	    // Counter hanya jalan saat tidak sedang sequence reset/release
	    IF #SeqMco = 0 THEN
	        IF "Win".Msc.Mco.Act < "Win".Msc.Mco.Set THEN
	            "Win".Msc.Mco.Act := "Win".Msc.Mco.Act + #McoStep;

	            IF "Win".Msc.Mco.Act >= "Win".Msc.Mco.Set THEN
	                "Win".Msc.Mco.Act := "Win".Msc.Mco.Set;
	                #McoReachedLatch := TRUE;
	            END_IF;
	        END_IF;
	    END_IF;

	    // Remaining meter
	    #McoRemain := "Win".Msc.Mco.Set - "Win".Msc.Mco.Act;
	    IF #McoRemain < 0.0 THEN
	        #McoRemain := 0.0;
	    END_IF;

	    // Time remaining dalam menit
	    IF #LineSpd > 0.0 THEN
	        "Win".Msc.Mco.Tim := #McoRemain / #LineSpd;
	    ELSE
	        "Win".Msc.Mco.Tim := 0.0;
	    END_IF;

	    // Trigger sequence jika setpoint tercapai
	    IF (#McoReachedLatch) AND (#SeqMco = 0) THEN
	        #McoReachedLatch := FALSE;
	        #SeqMco := 1;
	    END_IF;

	    // Sequential pulse:
	    // step 1 : Rst TRUE
	    // step 2 : Rst FALSE, Rel TRUE, reset Act ke 0
	    // step 0 : semua FALSE
	    CASE #SeqMco OF
	        0:
	            ;
	        1:
	            "Win".Msc.Mco.Rst := TRUE;
	            #SeqMco := 2;

	        2:
	            "Win".Msc.Mco.Rel := TRUE;
	            "Win".Msc.Mco.Act := 0.0;
	            #SeqMco := 0;
	        ELSE
	            #SeqMco := 0;
	    END_CASE;

	    "Win".Msc.AutCycTim.Act := "FC_NoiseReal"(Base := 300.0, Amp := #Amp_PosMm, Lo := #Lo, Hi := #Hi, Seed := #Seed);

	    // =========================
	    // WINDER 1 & 2
	    // =========================
	    "Win".W01.Drv.SpdSet := "FC_NoiseReal"(Base := 177.7, Amp := #Amp_SpdMpm, Lo := #Lo, Hi := #Hi, Seed := #Seed);
	    "Win".W01.Drv.SpdAct := "FC_NoiseReal"(Base := 171.2, Amp := #Amp_SpdMpm, Lo := #Lo, Hi := #Hi, Seed := #Seed);
	    "Win".W01.Drv.LoaAct := "FC_NoiseReal"(Base := 10.3, Amp := #Amp_LoaPct, Lo := #Lo, Hi := #Hi, Seed := #Seed);
	    "Win".W01.Gbl.TenSet := "FC_NoiseReal"(Base := 232.4, Amp := #Amp_TenNm, Lo := #Lo, Hi := #Hi, Seed := #Seed);
	    "Win".W01.Gbl.ScwTenSet := "FC_NoiseReal"(Base := 15.0, Amp := #Amp_LoaPct, Lo := #Lo, Hi := #Hi, Seed := #Seed);
	    "Win".W01.Prs.SetAct := "FC_NoiseReal"(Base := 1059.0, Amp := #Amp_PrsN, Lo := #Lo, Hi := #Hi, Seed := #Seed);
	    "Win".W01.Dia.Act := "FC_NoiseReal"(Base := 576.0, Amp := #Amp_PosMm, Lo := #Lo, Hi := #Hi, Seed := #Seed);

	    "Win".W02.Drv.SpdSet := "FC_NoiseReal"(Base := 0.0, Amp := #Amp_SpdMpm, Lo := #Lo, Hi := #Hi, Seed := #Seed);
	    "Win".W02.Drv.SpdAct := "FC_NoiseReal"(Base := 0.0, Amp := #Amp_SpdMpm, Lo := #Lo, Hi := #Hi, Seed := #Seed);
	    "Win".W02.Drv.LoaAct := "FC_NoiseReal"(Base := 0.0, Amp := #Amp_LoaPct, Lo := #Lo, Hi := #Hi, Seed := #Seed);
	    "Win".W02.Gbl.TenSet := "FC_NoiseReal"(Base := 234.4, Amp := #Amp_TenNm, Lo := #Lo, Hi := #Hi, Seed := #Seed);
	    "Win".W02.Gbl.ScwTenSet := "FC_NoiseReal"(Base := 15.0, Amp := #Amp_LoaPct, Lo := #Lo, Hi := #Hi, Seed := #Seed);
	    "Win".W02.Prs.SetAct := "FC_NoiseReal"(Base := 1056.0, Amp := #Amp_PrsN, Lo := #Lo, Hi := #Hi, Seed := #Seed);
	    "Win".W02.Dia.Act := "FC_NoiseReal"(Base := 0.0, Amp := #Amp_PosMm, Lo := #Lo, Hi := #Hi, Seed := #Seed);

END_FUNCTION_BLOCK

FUNCTION "FC_Fluct_DB325_StrTdoOut" : Void
{ S7_Optimized_Access := 'TRUE' }
VERSION : 0.1
// ============================================================
// FLUCTUATION DB325 (StrTdoOut) - TDO Outlet
// ============================================================
   VAR_INPUT
      Enable : Bool;   // amplitudo fluktuasi
      Amp_TmpC : Real;   // Â±Â°C
      Amp_Y_Pct : Real;   // Â±%
      Amp_SpdMpm : Real;   // Â± m/min
      Amp_Loa_Pct : Real;   // Â± %
   END_VAR

   VAR_IN_OUT
      Seed : DInt;
   END_VAR

   VAR_TEMP
      Lo : Real;
      Hi : Real;
   END_VAR


BEGIN
	    IF NOT #Enable THEN
	        RETURN;
	    END_IF;

	    #Lo := -3.4E38;
	    #Hi := 3.4E38;

	    // -------------------------
	    // Drive TDO Outlet (Drv001)
	    // -------------------------
	    "StrTdoOut".Drv001.SpdSet := "FC_NoiseReal"(Base := 175.0, Amp := #Amp_SpdMpm, Lo := #Lo, Hi := #Hi, Seed := #Seed);
	    "StrTdoOut".Drv001.SpdAct := "FC_NoiseReal"(Base := 175.0, Amp := #Amp_SpdMpm, Lo := #Lo, Hi := #Hi, Seed := #Seed);
	    "StrTdoOut".Drv001.LoaAct := "FC_NoiseReal"(Base := 20.8, Amp := #Amp_Loa_Pct, Lo := #Lo, Hi := #Hi, Seed := #Seed);

	    // -------------------------
	    // All Zone
	    // -------------------------
	    "StrTdoOut".TmpAll.Set := "FC_NoiseReal"(Base := 145.0, Amp := #Amp_TmpC, Lo := #Lo, Hi := #Hi, Seed := #Seed);

	    // -------------------------
	    // Annealing 1.1 (Ann011)
	    // -------------------------
	    "StrTdoOut".TmpAnn011.Set := "FC_NoiseReal"(Base := 145.0, Amp := #Amp_TmpC, Lo := #Lo, Hi := #Hi, Seed := #Seed);
	    "StrTdoOut".TmpAnn011.Act := "FC_NoiseReal"(Base := 145.1, Amp := #Amp_TmpC, Lo := #Lo, Hi := #Hi, Seed := #Seed);
	    "StrTdoOut".TmpAnn011.Y := "FC_NoiseReal"(Base := 0.0, Amp := #Amp_Y_Pct, Lo := #Lo, Hi := #Hi, Seed := #Seed);

	    // Annealing 1.2 (Ann012)
	    "StrTdoOut".TmpAnn012.Set := "FC_NoiseReal"(Base := 145.0, Amp := #Amp_TmpC, Lo := #Lo, Hi := #Hi, Seed := #Seed);
	    "StrTdoOut".TmpAnn012.Act := "FC_NoiseReal"(Base := 148.1, Amp := #Amp_TmpC, Lo := #Lo, Hi := #Hi, Seed := #Seed);
	    "StrTdoOut".TmpAnn012.Y := "FC_NoiseReal"(Base := 0.0, Amp := #Amp_Y_Pct, Lo := #Lo, Hi := #Hi, Seed := #Seed);

	    // -------------------------
	    // Annealing 2.1 (Ann021)
	    // -------------------------
	    "StrTdoOut".TmpAnn021.Set := "FC_NoiseReal"(Base := 135.0, Amp := #Amp_TmpC, Lo := #Lo, Hi := #Hi, Seed := #Seed);
	    "StrTdoOut".TmpAnn021.Act := "FC_NoiseReal"(Base := 134.7, Amp := #Amp_TmpC, Lo := #Lo, Hi := #Hi, Seed := #Seed);
	    "StrTdoOut".TmpAnn021.Y := "FC_NoiseReal"(Base := 3.0, Amp := #Amp_Y_Pct, Lo := #Lo, Hi := #Hi, Seed := #Seed);

	    // Annealing 2.2 (Ann022)
	    "StrTdoOut".TmpAnn022.Set := "FC_NoiseReal"(Base := 135.0, Amp := #Amp_TmpC, Lo := #Lo, Hi := #Hi, Seed := #Seed);
	    "StrTdoOut".TmpAnn022.Act := "FC_NoiseReal"(Base := 136.2, Amp := #Amp_TmpC, Lo := #Lo, Hi := #Hi, Seed := #Seed);
	    "StrTdoOut".TmpAnn022.Y := "FC_NoiseReal"(Base := 0.0, Amp := #Amp_Y_Pct, Lo := #Lo, Hi := #Hi, Seed := #Seed);

	    // -------------------------
	    // Annealing 3.1 (Ann031)
	    // -------------------------
	    "StrTdoOut".TmpAnn031.Set := "FC_NoiseReal"(Base := 135.0, Amp := #Amp_TmpC, Lo := #Lo, Hi := #Hi, Seed := #Seed);
	    "StrTdoOut".TmpAnn031.Act := "FC_NoiseReal"(Base := 135.1, Amp := #Amp_TmpC, Lo := #Lo, Hi := #Hi, Seed := #Seed);
	    "StrTdoOut".TmpAnn031.Y := "FC_NoiseReal"(Base := 8.0, Amp := #Amp_Y_Pct, Lo := #Lo, Hi := #Hi, Seed := #Seed);

	    // Annealing 3.2 (Ann032)
	    "StrTdoOut".TmpAnn032.Set := "FC_NoiseReal"(Base := 135.0, Amp := #Amp_TmpC, Lo := #Lo, Hi := #Hi, Seed := #Seed);
	    "StrTdoOut".TmpAnn032.Act := "FC_NoiseReal"(Base := 133.5, Amp := #Amp_TmpC, Lo := #Lo, Hi := #Hi, Seed := #Seed);
	    "StrTdoOut".TmpAnn032.Y := "FC_NoiseReal"(Base := 11.0, Amp := #Amp_Y_Pct, Lo := #Lo, Hi := #Hi, Seed := #Seed);

END_FUNCTION

FUNCTION "FC_Fluct_DB323_324_TdoInlMid" : Void
{ S7_Optimized_Access := 'TRUE' }
VERSION : 0.1
// ============================================================
// FLUCTUATION DB323 + DB324
// AREA: StrTdoInl + StrTdoMid
// ============================================================
   VAR_INPUT
      Enable : Bool;   // amplitudo fluktuasi
      Amp_TmpC : Real;   // Â±Â°C
      Amp_Y_Pct : Real;   // Â±%
   END_VAR

   VAR_IN_OUT
      Seed : DInt;
   END_VAR

   VAR_TEMP
      Lo : Real;
      Hi : Real;
   END_VAR


BEGIN
	    IF NOT #Enable THEN
	        RETURN;
	    END_IF;

	    #Lo := -3.4E38;
	    #Hi := 3.4E38;

	    // =====================================================
	    // DB323 - StrTdoInl
	    // =====================================================

	    // All Zone
	    "StrTdoInl".TmpAll.Set := "FC_NoiseReal"(Base := 179.0, Amp := #Amp_TmpC, Lo := #Lo, Hi := #Hi, Seed := #Seed);

	    // Preheating 1
	    "StrTdoInl".TmpPrh001.Set := "FC_NoiseReal"(Base := 164.0, Amp := #Amp_TmpC, Lo := #Lo, Hi := #Hi, Seed := #Seed);
	    "StrTdoInl".TmpPrh001.Act := "FC_NoiseReal"(Base := 164.0, Amp := #Amp_TmpC, Lo := #Lo, Hi := #Hi, Seed := #Seed);
	    "StrTdoInl".TmpPrh001.Y := "FC_NoiseReal"(Base := 35.0, Amp := #Amp_Y_Pct, Lo := #Lo, Hi := #Hi, Seed := #Seed);

	    // Preheating 2
	    "StrTdoInl".TmpPrh002.Set := "FC_NoiseReal"(Base := 174.0, Amp := #Amp_TmpC, Lo := #Lo, Hi := #Hi, Seed := #Seed);
	    "StrTdoInl".TmpPrh002.Act := "FC_NoiseReal"(Base := 173.3, Amp := #Amp_TmpC, Lo := #Lo, Hi := #Hi, Seed := #Seed);
	    "StrTdoInl".TmpPrh002.Y := "FC_NoiseReal"(Base := 100.0, Amp := #Amp_Y_Pct, Lo := #Lo, Hi := #Hi, Seed := #Seed);

	    // Preheating 3
	    "StrTdoInl".TmpPrh003.Set := "FC_NoiseReal"(Base := 179.0, Amp := #Amp_TmpC, Lo := #Lo, Hi := #Hi, Seed := #Seed);
	    "StrTdoInl".TmpPrh003.Act := "FC_NoiseReal"(Base := 179.2, Amp := #Amp_TmpC, Lo := #Lo, Hi := #Hi, Seed := #Seed);
	    "StrTdoInl".TmpPrh003.Y := "FC_NoiseReal"(Base := 20.0, Amp := #Amp_Y_Pct, Lo := #Lo, Hi := #Hi, Seed := #Seed);

	    // =====================================================
	    // DB324 - StrTdoMid
	    // =====================================================

	    // All Zone
	    "StrTdoMid".TmpAll.Set := "FC_NoiseReal"(Base := 157.0, Amp := #Amp_TmpC, Lo := #Lo, Hi := #Hi, Seed := #Seed);

	    // Drawing 1.1
	    "StrTdoMid".TmpDrw011.Set := "FC_NoiseReal"(Base := 157.0, Amp := #Amp_TmpC, Lo := #Lo, Hi := #Hi, Seed := #Seed);
	    "StrTdoMid".TmpDrw011.Act := "FC_NoiseReal"(Base := 157.0, Amp := #Amp_TmpC, Lo := #Lo, Hi := #Hi, Seed := #Seed);
	    "StrTdoMid".TmpDrw011.Y := "FC_NoiseReal"(Base := 54.0, Amp := #Amp_Y_Pct, Lo := #Lo, Hi := #Hi, Seed := #Seed);

	    // Drawing 1.2
	    "StrTdoMid".TmpDrw012.Set := "FC_NoiseReal"(Base := 157.0, Amp := #Amp_TmpC, Lo := #Lo, Hi := #Hi, Seed := #Seed);
	    "StrTdoMid".TmpDrw012.Act := "FC_NoiseReal"(Base := 156.8, Amp := #Amp_TmpC, Lo := #Lo, Hi := #Hi, Seed := #Seed);
	    "StrTdoMid".TmpDrw012.Y := "FC_NoiseReal"(Base := 14.0, Amp := #Amp_Y_Pct, Lo := #Lo, Hi := #Hi, Seed := #Seed);

	    // Drawing 2.1
	    "StrTdoMid".TmpDrw021.Set := "FC_NoiseReal"(Base := 157.0, Amp := #Amp_TmpC, Lo := #Lo, Hi := #Hi, Seed := #Seed);
	    "StrTdoMid".TmpDrw021.Act := "FC_NoiseReal"(Base := 156.9, Amp := #Amp_TmpC, Lo := #Lo, Hi := #Hi, Seed := #Seed);
	    "StrTdoMid".TmpDrw021.Y := "FC_NoiseReal"(Base := 4.0, Amp := #Amp_Y_Pct, Lo := #Lo, Hi := #Hi, Seed := #Seed);

	    // Drawing 2.2
	    "StrTdoMid".TmpDrw022.Set := "FC_NoiseReal"(Base := 157.0, Amp := #Amp_TmpC, Lo := #Lo, Hi := #Hi, Seed := #Seed);
	    "StrTdoMid".TmpDrw022.Act := "FC_NoiseReal"(Base := 157.0, Amp := #Amp_TmpC, Lo := #Lo, Hi := #Hi, Seed := #Seed);
	    "StrTdoMid".TmpDrw022.Y := "FC_NoiseReal"(Base := 2.0, Amp := #Amp_Y_Pct, Lo := #Lo, Hi := #Hi, Seed := #Seed);

	    // Drawing 3.1
	    "StrTdoMid".TmpDrw031.Set := "FC_NoiseReal"(Base := 156.0, Amp := #Amp_TmpC, Lo := #Lo, Hi := #Hi, Seed := #Seed);
	    "StrTdoMid".TmpDrw031.Act := "FC_NoiseReal"(Base := 156.0, Amp := #Amp_TmpC, Lo := #Lo, Hi := #Hi, Seed := #Seed);
	    "StrTdoMid".TmpDrw031.Y := "FC_NoiseReal"(Base := 63.0, Amp := #Amp_Y_Pct, Lo := #Lo, Hi := #Hi, Seed := #Seed);

	    // Drawing 3.2
	    "StrTdoMid".TmpDrw032.Set := "FC_NoiseReal"(Base := 156.0, Amp := #Amp_TmpC, Lo := #Lo, Hi := #Hi, Seed := #Seed);
	    "StrTdoMid".TmpDrw032.Act := "FC_NoiseReal"(Base := 155.8, Amp := #Amp_TmpC, Lo := #Lo, Hi := #Hi, Seed := #Seed);
	    "StrTdoMid".TmpDrw032.Y := "FC_NoiseReal"(Base := 10.0, Amp := #Amp_Y_Pct, Lo := #Lo, Hi := #Hi, Seed := #Seed);

	    // Drawing 4.1
	    "StrTdoMid".TmpDrw041.Set := "FC_NoiseReal"(Base := 155.0, Amp := #Amp_TmpC, Lo := #Lo, Hi := #Hi, Seed := #Seed);
	    "StrTdoMid".TmpDrw041.Act := "FC_NoiseReal"(Base := 154.3, Amp := #Amp_TmpC, Lo := #Lo, Hi := #Hi, Seed := #Seed);
	    "StrTdoMid".TmpDrw041.Y := "FC_NoiseReal"(Base := 3.0, Amp := #Amp_Y_Pct, Lo := #Lo, Hi := #Hi, Seed := #Seed);

	    // Drawing 4.2
	    "StrTdoMid".TmpDrw042.Set := "FC_NoiseReal"(Base := 155.0, Amp := #Amp_TmpC, Lo := #Lo, Hi := #Hi, Seed := #Seed);
	    "StrTdoMid".TmpDrw042.Act := "FC_NoiseReal"(Base := 156.0, Amp := #Amp_TmpC, Lo := #Lo, Hi := #Hi, Seed := #Seed);
	    "StrTdoMid".TmpDrw042.Y := "FC_NoiseReal"(Base := 0.0, Amp := #Amp_Y_Pct, Lo := #Lo, Hi := #Hi, Seed := #Seed);

END_FUNCTION

FUNCTION "FC_Fluct_DB313_ExtFil" : Void
{ S7_Optimized_Access := 'TRUE' }
VERSION : 0.1
// ============================================================
// FLUCTUATION DB313 (ExtFil)
// ============================================================
   VAR_INPUT
      Enable : Bool;   // amplitudo fluktuasi
      Amp_TmpC : Real;   // Â±Â°C
      Amp_PrsBar : Real;   // Â±bar
      Amp_Y_Pct : Real;   // Â±%
   END_VAR

   VAR_IN_OUT
      Seed : DInt;
   END_VAR

   VAR_TEMP
      Lo : Real;
      Hi : Real;
   END_VAR


BEGIN
	    IF NOT #Enable THEN
	        RETURN;
	    END_IF;

	    #Lo := -3.4E38;
	    #Hi := 3.4E38;

	    // =========================
	    // Pressure (S7_PRS) - base dari gambar + comment ExtFil.db
	    // Prs001: before filter  (Press P3 = 97.9 bar)
	    // Prs002: after filter   (Press P2 = 135.6 bar)
	    // Prs012: diff pressure  (Diff Press = 37.7 bar)
	    // Prs003: before die     (Press P4 = 0.0 bar)
	    // =========================
	    "ExtFil".Prs001.Act := "FC_NoiseReal"(Base := 97.9, Amp := #Amp_PrsBar, Lo := #Lo, Hi := #Hi, Seed := #Seed);
	    "ExtFil".Prs002.Act := "FC_NoiseReal"(Base := 135.6, Amp := #Amp_PrsBar, Lo := #Lo, Hi := #Hi, Seed := #Seed);
	    "ExtFil".Prs012.Act := "FC_NoiseReal"(Base := 37.7, Amp := #Amp_PrsBar, Lo := #Lo, Hi := #Hi, Seed := #Seed);
	    "ExtFil".Prs003.Act := "FC_NoiseReal"(Base := 0.0, Amp := #Amp_PrsBar, Lo := #Lo, Hi := #Hi, Seed := #Seed);

	    // =========================
	    // Melt Temp (S7_ACT) - base dari gambar
	    // TmpMel001: before filter (Melt Temp T3 = 241.1 Â°C)
	    // TmpMel002: after filter  (Melt Temp T2 = 244.6 Â°C)
	    // TmpMel003: before die    (Melt Temp T4 = 1999.9 Â°C)  // sesuai tampilan
	    // TmpMel004: preheating filter (Pre.Filter = 32.4 Â°C)
	    // =========================
	    "ExtFil".TmpMel001.Act := "FC_NoiseReal"(Base := 241.1, Amp := #Amp_TmpC, Lo := #Lo, Hi := #Hi, Seed := #Seed);
	    "ExtFil".TmpMel002.Act := "FC_NoiseReal"(Base := 244.6, Amp := #Amp_TmpC, Lo := #Lo, Hi := #Hi, Seed := #Seed);
	    "ExtFil".TmpMel003.Act := "FC_NoiseReal"(Base := 1999.9, Amp := #Amp_TmpC, Lo := #Lo, Hi := #Hi, Seed := #Seed);
	    "ExtFil".TmpMel004.Act := "FC_NoiseReal"(Base := 32.4, Amp := #Amp_TmpC, Lo := #Lo, Hi := #Hi, Seed := #Seed);

	    // =========================
	    // All Zone
	    // =========================
	    "ExtFil".TmpAll.Set := "FC_NoiseReal"(Base := 235.0, Amp := #Amp_TmpC, Lo := #Lo, Hi := #Hi, Seed := #Seed);

	    // =========================
	    // Adapter / Pipe / Filter (CTL_GEN): .Act / .Set / .Y
	    // =========================

	    // Adapter (kanan)
	    "ExtFil".TmpAdp.Set := "FC_NoiseReal"(Base := 235.0, Amp := #Amp_TmpC, Lo := #Lo, Hi := #Hi, Seed := #Seed);
	    "ExtFil".TmpAdp.Act := "FC_NoiseReal"(Base := 235.0, Amp := #Amp_TmpC, Lo := #Lo, Hi := #Hi, Seed := #Seed);
	    "ExtFil".TmpAdp.Y := "FC_NoiseReal"(Base := 39.0, Amp := #Amp_Y_Pct, Lo := #Lo, Hi := #Hi, Seed := #Seed);

	    // Adapter 1 (bawah kanan)
	    "ExtFil".TmpAdp001.Set := "FC_NoiseReal"(Base := 235.0, Amp := #Amp_TmpC, Lo := #Lo, Hi := #Hi, Seed := #Seed);
	    "ExtFil".TmpAdp001.Act := "FC_NoiseReal"(Base := 235.0, Amp := #Amp_TmpC, Lo := #Lo, Hi := #Hi, Seed := #Seed);
	    "ExtFil".TmpAdp001.Y := "FC_NoiseReal"(Base := 31.0, Amp := #Amp_Y_Pct, Lo := #Lo, Hi := #Hi, Seed := #Seed);

	    // Adapter 2 (bawah kiri)
	    "ExtFil".TmpAdp002.Set := "FC_NoiseReal"(Base := 235.0, Amp := #Amp_TmpC, Lo := #Lo, Hi := #Hi, Seed := #Seed);
	    "ExtFil".TmpAdp002.Act := "FC_NoiseReal"(Base := 235.1, Amp := #Amp_TmpC, Lo := #Lo, Hi := #Hi, Seed := #Seed);
	    "ExtFil".TmpAdp002.Y := "FC_NoiseReal"(Base := 45.0, Amp := #Amp_Y_Pct, Lo := #Lo, Hi := #Hi, Seed := #Seed);

	    // Pipe 2.1 .. 2.4
	    "ExtFil".TmpPip021.Set := "FC_NoiseReal"(Base := 235.0, Amp := #Amp_TmpC, Lo := #Lo, Hi := #Hi, Seed := #Seed);
	    "ExtFil".TmpPip021.Act := "FC_NoiseReal"(Base := 235.0, Amp := #Amp_TmpC, Lo := #Lo, Hi := #Hi, Seed := #Seed);
	    "ExtFil".TmpPip021.Y := "FC_NoiseReal"(Base := 62.0, Amp := #Amp_Y_Pct, Lo := #Lo, Hi := #Hi, Seed := #Seed);

	    "ExtFil".TmpPip022.Set := "FC_NoiseReal"(Base := 235.0, Amp := #Amp_TmpC, Lo := #Lo, Hi := #Hi, Seed := #Seed);
	    "ExtFil".TmpPip022.Act := "FC_NoiseReal"(Base := 234.9, Amp := #Amp_TmpC, Lo := #Lo, Hi := #Hi, Seed := #Seed);
	    "ExtFil".TmpPip022.Y := "FC_NoiseReal"(Base := 16.0, Amp := #Amp_Y_Pct, Lo := #Lo, Hi := #Hi, Seed := #Seed);

	    "ExtFil".TmpPip023.Set := "FC_NoiseReal"(Base := 235.0, Amp := #Amp_TmpC, Lo := #Lo, Hi := #Hi, Seed := #Seed);
	    "ExtFil".TmpPip023.Act := "FC_NoiseReal"(Base := 235.2, Amp := #Amp_TmpC, Lo := #Lo, Hi := #Hi, Seed := #Seed);
	    "ExtFil".TmpPip023.Y := "FC_NoiseReal"(Base := 90.0, Amp := #Amp_Y_Pct, Lo := #Lo, Hi := #Hi, Seed := #Seed);

	    "ExtFil".TmpPip024.Set := "FC_NoiseReal"(Base := 235.0, Amp := #Amp_TmpC, Lo := #Lo, Hi := #Hi, Seed := #Seed);
	    "ExtFil".TmpPip024.Act := "FC_NoiseReal"(Base := 235.0, Amp := #Amp_TmpC, Lo := #Lo, Hi := #Hi, Seed := #Seed);
	    "ExtFil".TmpPip024.Y := "FC_NoiseReal"(Base := 36.0, Amp := #Amp_Y_Pct, Lo := #Lo, Hi := #Hi, Seed := #Seed);

	    // Filter 1..3
	    "ExtFil".TmpFil001.Set := "FC_NoiseReal"(Base := 255.0, Amp := #Amp_TmpC, Lo := #Lo, Hi := #Hi, Seed := #Seed);
	    "ExtFil".TmpFil001.Act := "FC_NoiseReal"(Base := 255.0, Amp := #Amp_TmpC, Lo := #Lo, Hi := #Hi, Seed := #Seed);
	    "ExtFil".TmpFil001.Y := "FC_NoiseReal"(Base := 16.0, Amp := #Amp_Y_Pct, Lo := #Lo, Hi := #Hi, Seed := #Seed);

	    "ExtFil".TmpFil002.Set := "FC_NoiseReal"(Base := 255.0, Amp := #Amp_TmpC, Lo := #Lo, Hi := #Hi, Seed := #Seed);
	    "ExtFil".TmpFil002.Act := "FC_NoiseReal"(Base := 255.1, Amp := #Amp_TmpC, Lo := #Lo, Hi := #Hi, Seed := #Seed);
	    "ExtFil".TmpFil002.Y := "FC_NoiseReal"(Base := 20.0, Amp := #Amp_Y_Pct, Lo := #Lo, Hi := #Hi, Seed := #Seed);

	    "ExtFil".TmpFil003.Set := "FC_NoiseReal"(Base := 235.0, Amp := #Amp_TmpC, Lo := #Lo, Hi := #Hi, Seed := #Seed);
	    "ExtFil".TmpFil003.Act := "FC_NoiseReal"(Base := 235.2, Amp := #Amp_TmpC, Lo := #Lo, Hi := #Hi, Seed := #Seed);
	    "ExtFil".TmpFil003.Y := "FC_NoiseReal"(Base := 14.0, Amp := #Amp_Y_Pct, Lo := #Lo, Hi := #Hi, Seed := #Seed);

	    // Pipe 3.1 .. 3.5
	    "ExtFil".TmpPip031.Set := "FC_NoiseReal"(Base := 235.0, Amp := #Amp_TmpC, Lo := #Lo, Hi := #Hi, Seed := #Seed);
	    "ExtFil".TmpPip031.Act := "FC_NoiseReal"(Base := 235.1, Amp := #Amp_TmpC, Lo := #Lo, Hi := #Hi, Seed := #Seed);
	    "ExtFil".TmpPip031.Y := "FC_NoiseReal"(Base := 53.0, Amp := #Amp_Y_Pct, Lo := #Lo, Hi := #Hi, Seed := #Seed);

	    "ExtFil".TmpPip032.Set := "FC_NoiseReal"(Base := 235.0, Amp := #Amp_TmpC, Lo := #Lo, Hi := #Hi, Seed := #Seed);
	    "ExtFil".TmpPip032.Act := "FC_NoiseReal"(Base := 235.0, Amp := #Amp_TmpC, Lo := #Lo, Hi := #Hi, Seed := #Seed);
	    "ExtFil".TmpPip032.Y := "FC_NoiseReal"(Base := 9.0, Amp := #Amp_Y_Pct, Lo := #Lo, Hi := #Hi, Seed := #Seed);

	    "ExtFil".TmpPip033.Set := "FC_NoiseReal"(Base := 235.0, Amp := #Amp_TmpC, Lo := #Lo, Hi := #Hi, Seed := #Seed);
	    "ExtFil".TmpPip033.Act := "FC_NoiseReal"(Base := 235.0, Amp := #Amp_TmpC, Lo := #Lo, Hi := #Hi, Seed := #Seed);
	    "ExtFil".TmpPip033.Y := "FC_NoiseReal"(Base := 7.0, Amp := #Amp_Y_Pct, Lo := #Lo, Hi := #Hi, Seed := #Seed);

	    "ExtFil".TmpPip034.Set := "FC_NoiseReal"(Base := 235.0, Amp := #Amp_TmpC, Lo := #Lo, Hi := #Hi, Seed := #Seed);
	    "ExtFil".TmpPip034.Act := "FC_NoiseReal"(Base := 235.0, Amp := #Amp_TmpC, Lo := #Lo, Hi := #Hi, Seed := #Seed);
	    "ExtFil".TmpPip034.Y := "FC_NoiseReal"(Base := 10.0, Amp := #Amp_Y_Pct, Lo := #Lo, Hi := #Hi, Seed := #Seed);

	    "ExtFil".TmpPip035.Set := "FC_NoiseReal"(Base := 235.0, Amp := #Amp_TmpC, Lo := #Lo, Hi := #Hi, Seed := #Seed);
	    "ExtFil".TmpPip035.Act := "FC_NoiseReal"(Base := 235.0, Amp := #Amp_TmpC, Lo := #Lo, Hi := #Hi, Seed := #Seed);
	    "ExtFil".TmpPip035.Y := "FC_NoiseReal"(Base := 76.0, Amp := #Amp_Y_Pct, Lo := #Lo, Hi := #Hi, Seed := #Seed);

END_FUNCTION

FUNCTION "FC_Fluct_DB322_StrMdo" : Void
{ S7_Optimized_Access := 'TRUE' }
VERSION : 0.1
// ============================================================
// FLUCTUATION DB322 (StrMdo) - MDO
// ============================================================
   VAR_INPUT
      Enable : Bool;   // amplitudo fluktuasi
      Amp_TmpC : Real;   // Â±Â°C
      Amp_Y_Pct : Real;   // Â±% drive speed & load
      Amp_SpdMpm : Real;   // Â± m/min
      Amp_LoaPct : Real;   // Â± %
   END_VAR

   VAR_IN_OUT
      Seed : DInt;
   END_VAR

   VAR_TEMP
      Lo : Real;
      Hi : Real;
   END_VAR


BEGIN
	    IF NOT #Enable THEN
	        RETURN;
	    END_IF;

	    #Lo := -3.4E38;
	    #Hi := 3.4E38;

	    // =========================
	    // Drives (instruksi kamu)
	    // =========================
	    // MDO 1
	    "StrMdo".Drv001.SpdSet := "FC_NoiseReal"(Base := 28.0, Amp := #Amp_SpdMpm, Lo := #Lo, Hi := #Hi, Seed := #Seed);
	    "StrMdo".Drv001.SpdAct := "FC_NoiseReal"(Base := 28.4, Amp := #Amp_SpdMpm, Lo := #Lo, Hi := #Hi, Seed := #Seed);
	    "StrMdo".Drv001.LoaAct := "FC_NoiseReal"(Base := -13.5, Amp := #Amp_LoaPct, Lo := #Lo, Hi := #Hi, Seed := #Seed);

	    // MDO 2 (SpdSet tidak tampil di layar â†’ disamakan dengan Act)
	    "StrMdo".Drv002.SpdSet := "FC_NoiseReal"(Base := 159.0, Amp := #Amp_SpdMpm, Lo := #Lo, Hi := #Hi, Seed := #Seed);
	    "StrMdo".Drv002.SpdAct := "FC_NoiseReal"(Base := 159.0, Amp := #Amp_SpdMpm, Lo := #Lo, Hi := #Hi, Seed := #Seed);
	    "StrMdo".Drv002.LoaAct := "FC_NoiseReal"(Base := 5.5, Amp := #Amp_LoaPct, Lo := #Lo, Hi := #Hi, Seed := #Seed);

	    // MDO 3 (SpdSet tidak tampil di layar â†’ disamakan dengan Act)
	    "StrMdo".Drv003.SpdSet := "FC_NoiseReal"(Base := 171.0, Amp := #Amp_SpdMpm, Lo := #Lo, Hi := #Hi, Seed := #Seed);
	    "StrMdo".Drv003.SpdAct := "FC_NoiseReal"(Base := 171.0, Amp := #Amp_SpdMpm, Lo := #Lo, Hi := #Hi, Seed := #Seed);
	    "StrMdo".Drv003.LoaAct := "FC_NoiseReal"(Base := 12.1, Amp := #Amp_LoaPct, Lo := #Lo, Hi := #Hi, Seed := #Seed);

	    // Auxiliary Winder (DrvAuw)
	    "StrMdo".DrvAuw.SpdSet := "FC_NoiseReal"(Base := 0.0, Amp := #Amp_SpdMpm, Lo := #Lo, Hi := #Hi, Seed := #Seed);
	    "StrMdo".DrvAuw.SpdAct := "FC_NoiseReal"(Base := 0.0, Amp := #Amp_SpdMpm, Lo := #Lo, Hi := #Hi, Seed := #Seed);
	    "StrMdo".DrvAuw.LoaAct := "FC_NoiseReal"(Base := 0.0, Amp := #Amp_LoaPct, Lo := #Lo, Hi := #Hi, Seed := #Seed);

	    // =========================
	    // All Zone (ambil set tertinggi yg dominan di MDO: 114.0Â°C)
	    // =========================
	    "StrMdo".TmpAll.Set := "FC_NoiseReal"(Base := 114.0, Amp := #Amp_TmpC, Lo := #Lo, Hi := #Hi, Seed := #Seed);

	    // =========================
	    // Preheating 1..5
	    // =========================
	    "StrMdo".TmpPrh001.Set := "FC_NoiseReal"(Base := 112.0, Amp := #Amp_TmpC, Lo := #Lo, Hi := #Hi, Seed := #Seed);
	    "StrMdo".TmpPrh001.Act := "FC_NoiseReal"(Base := 112.2, Amp := #Amp_TmpC, Lo := #Lo, Hi := #Hi, Seed := #Seed);
	    "StrMdo".TmpPrh001.Y := "FC_NoiseReal"(Base := 1.0, Amp := #Amp_Y_Pct, Lo := #Lo, Hi := #Hi, Seed := #Seed);

	    "StrMdo".TmpPrh002.Set := "FC_NoiseReal"(Base := 112.0, Amp := #Amp_TmpC, Lo := #Lo, Hi := #Hi, Seed := #Seed);
	    "StrMdo".TmpPrh002.Act := "FC_NoiseReal"(Base := 112.0, Amp := #Amp_TmpC, Lo := #Lo, Hi := #Hi, Seed := #Seed);
	    "StrMdo".TmpPrh002.Y := "FC_NoiseReal"(Base := 7.0, Amp := #Amp_Y_Pct, Lo := #Lo, Hi := #Hi, Seed := #Seed);

	    "StrMdo".TmpPrh003.Set := "FC_NoiseReal"(Base := 113.0, Amp := #Amp_TmpC, Lo := #Lo, Hi := #Hi, Seed := #Seed);
	    "StrMdo".TmpPrh003.Act := "FC_NoiseReal"(Base := 113.0, Amp := #Amp_TmpC, Lo := #Lo, Hi := #Hi, Seed := #Seed);
	    "StrMdo".TmpPrh003.Y := "FC_NoiseReal"(Base := 0.0, Amp := #Amp_Y_Pct, Lo := #Lo, Hi := #Hi, Seed := #Seed);

	    "StrMdo".TmpPrh004.Set := "FC_NoiseReal"(Base := 114.0, Amp := #Amp_TmpC, Lo := #Lo, Hi := #Hi, Seed := #Seed);
	    "StrMdo".TmpPrh004.Act := "FC_NoiseReal"(Base := 114.1, Amp := #Amp_TmpC, Lo := #Lo, Hi := #Hi, Seed := #Seed);
	    "StrMdo".TmpPrh004.Y := "FC_NoiseReal"(Base := 33.0, Amp := #Amp_Y_Pct, Lo := #Lo, Hi := #Hi, Seed := #Seed);

	    "StrMdo".TmpPrh005.Set := "FC_NoiseReal"(Base := 114.0, Amp := #Amp_TmpC, Lo := #Lo, Hi := #Hi, Seed := #Seed);
	    "StrMdo".TmpPrh005.Act := "FC_NoiseReal"(Base := 114.1, Amp := #Amp_TmpC, Lo := #Lo, Hi := #Hi, Seed := #Seed);
	    "StrMdo".TmpPrh005.Y := "FC_NoiseReal"(Base := 1.0, Amp := #Amp_Y_Pct, Lo := #Lo, Hi := #Hi, Seed := #Seed);

	    // =========================
	    // Drawing 1..3
	    // =========================
	    "StrMdo".TmpDrw001.Set := "FC_NoiseReal"(Base := 73.0, Amp := #Amp_TmpC, Lo := #Lo, Hi := #Hi, Seed := #Seed);
	    "StrMdo".TmpDrw001.Act := "FC_NoiseReal"(Base := 73.2, Amp := #Amp_TmpC, Lo := #Lo, Hi := #Hi, Seed := #Seed);
	    "StrMdo".TmpDrw001.Y := "FC_NoiseReal"(Base := -13.0, Amp := #Amp_Y_Pct, Lo := #Lo, Hi := #Hi, Seed := #Seed);

	    "StrMdo".TmpDrw002.Set := "FC_NoiseReal"(Base := 75.0, Amp := #Amp_TmpC, Lo := #Lo, Hi := #Hi, Seed := #Seed);
	    "StrMdo".TmpDrw002.Act := "FC_NoiseReal"(Base := 75.0, Amp := #Amp_TmpC, Lo := #Lo, Hi := #Hi, Seed := #Seed);
	    "StrMdo".TmpDrw002.Y := "FC_NoiseReal"(Base := -22.0, Amp := #Amp_Y_Pct, Lo := #Lo, Hi := #Hi, Seed := #Seed);

	    "StrMdo".TmpDrw003.Set := "FC_NoiseReal"(Base := 80.0, Amp := #Amp_TmpC, Lo := #Lo, Hi := #Hi, Seed := #Seed);
	    "StrMdo".TmpDrw003.Act := "FC_NoiseReal"(Base := 80.2, Amp := #Amp_TmpC, Lo := #Lo, Hi := #Hi, Seed := #Seed);
	    "StrMdo".TmpDrw003.Y := "FC_NoiseReal"(Base := -13.0, Amp := #Amp_Y_Pct, Lo := #Lo, Hi := #Hi, Seed := #Seed);

	    // =========================
	    // Annealing 1..2
	    // =========================
	    "StrMdo".TmpAnn001.Set := "FC_NoiseReal"(Base := 75.0, Amp := #Amp_TmpC, Lo := #Lo, Hi := #Hi, Seed := #Seed);
	    "StrMdo".TmpAnn001.Act := "FC_NoiseReal"(Base := 74.9, Amp := #Amp_TmpC, Lo := #Lo, Hi := #Hi, Seed := #Seed);
	    "StrMdo".TmpAnn001.Y := "FC_NoiseReal"(Base := -13.0, Amp := #Amp_Y_Pct, Lo := #Lo, Hi := #Hi, Seed := #Seed);

	    "StrMdo".TmpAnn002.Set := "FC_NoiseReal"(Base := 75.0, Amp := #Amp_TmpC, Lo := #Lo, Hi := #Hi, Seed := #Seed);
	    "StrMdo".TmpAnn002.Act := "FC_NoiseReal"(Base := 75.2, Amp := #Amp_TmpC, Lo := #Lo, Hi := #Hi, Seed := #Seed);
	    "StrMdo".TmpAnn002.Y := "FC_NoiseReal"(Base := -22.0, Amp := #Amp_Y_Pct, Lo := #Lo, Hi := #Hi, Seed := #Seed);

END_FUNCTION

FUNCTION "FC_Fluct_DB321_StrCas" : Void
{ S7_Optimized_Access := 'TRUE' }
VERSION : 0.1
// ============================================================
// FLUCTUATION DB321 (StrCas) - Chill Roll
// ============================================================
   VAR_INPUT
      Enable : Bool;   // amplitudo fluktuasi
      Amp_SpdPct : Real;   // Â±%  (fan speed)
      Amp_PrsMbar : Real;   // Â±mbar
      Amp_TmpC : Real;   // Â±Â°C
      Amp_Y_Pct : Real;   // Â±% drive chill roll (m/min dan load %)
      Amp_SpdMpm : Real;   // Â± m/min
      Amp_LoaPct : Real;   // Â± %
   END_VAR

   VAR_IN_OUT
      Seed : DInt;
   END_VAR

   VAR_TEMP
      Lo : Real;
      Hi : Real;
   END_VAR


BEGIN
	    IF NOT #Enable THEN
	        RETURN;
	    END_IF;

	    #Lo := -3.4E38;
	    #Hi := 3.4E38;

	    // =========================
	    // Drive Chill Roll (ambil dari DrvChr.*)
	    // =========================
	    "StrCas".DrvChr.SpdSet := "FC_NoiseReal"(Base := 28.3, Amp := #Amp_SpdMpm, Lo := #Lo, Hi := #Hi, Seed := #Seed);
	    "StrCas".DrvChr.SpdAct := "FC_NoiseReal"(Base := 28.3, Amp := #Amp_SpdMpm, Lo := #Lo, Hi := #Hi, Seed := #Seed);
	    "StrCas".DrvChr.LoaAct := "FC_NoiseReal"(Base := 0.6, Amp := #Amp_LoaPct, Lo := #Lo, Hi := #Hi, Seed := #Seed);

	    // =========================
	    // Air Knife Fan
	    // =========================
	    "StrCas".FanAkn.SpdAct := "FC_NoiseReal"(Base := 82.0, Amp := #Amp_SpdPct, Lo := #Lo, Hi := #Hi, Seed := #Seed);

	    // =========================
	    // Pressure Air Knife (di layar hanya 0.0 mbar)
	    // =========================
	    "StrCas".PrsAkn.Set := "FC_NoiseReal"(Base := 0.0, Amp := #Amp_PrsMbar, Lo := #Lo, Hi := #Hi, Seed := #Seed);
	    "StrCas".PrsAkn.Act := "FC_NoiseReal"(Base := 0.0, Amp := #Amp_PrsMbar, Lo := #Lo, Hi := #Hi, Seed := #Seed);
	    "StrCas".PrsAkn.Y := "FC_NoiseReal"(Base := 0.0, Amp := #Amp_Y_Pct, Lo := #Lo, Hi := #Hi, Seed := #Seed);

	    // =========================
	    // All Zone (pakai setpoint utama Chill Roll)
	    // =========================
	    "StrCas".TmpAll.Set := "FC_NoiseReal"(Base := 35.0, Amp := #Amp_TmpC, Lo := #Lo, Hi := #Hi, Seed := #Seed);

	    // =========================
	    // Chill Roll Temperature
	    // =========================
	    "StrCas".TmpChr.Set := "FC_NoiseReal"(Base := 35.0, Amp := #Amp_TmpC, Lo := #Lo, Hi := #Hi, Seed := #Seed);
	    "StrCas".TmpChr.Act := "FC_NoiseReal"(Base := 35.0, Amp := #Amp_TmpC, Lo := #Lo, Hi := #Hi, Seed := #Seed);
	    "StrCas".TmpChr.Y := "FC_NoiseReal"(Base := -33.0, Amp := #Amp_Y_Pct, Lo := #Lo, Hi := #Hi, Seed := #Seed);

	    // =========================
	    // Water Bath Temperature
	    // =========================
	    "StrCas".TmpWba.Set := "FC_NoiseReal"(Base := 30.0, Amp := #Amp_TmpC, Lo := #Lo, Hi := #Hi, Seed := #Seed);
	    "StrCas".TmpWba.Act := "FC_NoiseReal"(Base := 31.4, Amp := #Amp_TmpC, Lo := #Lo, Hi := #Hi, Seed := #Seed);
	    "StrCas".TmpWba.Y := "FC_NoiseReal"(Base := -99.0, Amp := #Amp_Y_Pct, Lo := #Lo, Hi := #Hi, Seed := #Seed);

END_FUNCTION

FUNCTION "FC_Fluct_DB317_ExtCox002" : Void
{ S7_Optimized_Access := 'TRUE' }
VERSION : 0.1
// ============================================================
// FLUCTUATION DB317 (ExtCox002)
// ============================================================
   VAR_INPUT
      Enable : Bool;   // amplitudo fluktuasi
      Amp_PowKw : Real;   // Â±kW
      Amp_SpdRpm : Real;   // Â±rpm
      Amp_TmpC : Real;   // Â±Â°C
      Amp_PrsBar : Real;   // Â±bar
      Amp_Y_Pct : Real;   // Â±%
      Amp_LoaPct : Real;   // Â±%
   END_VAR

   VAR_IN_OUT
      Seed : DInt;
   END_VAR

   VAR_TEMP
      Lo : Real;
      Hi : Real;
   END_VAR


BEGIN
	    IF NOT #Enable THEN
	        RETURN;
	    END_IF;

	    #Lo := -3.4E38;
	    #Hi := 3.4E38;

	    // =========================
	    // Drive (panel kiri bawah)
	    // =========================
	    "ExtCox002".Drv001.TmpAct := "FC_NoiseReal"(Base := 60.6, Amp := #Amp_TmpC, Lo := #Lo, Hi := #Hi, Seed := #Seed);
	    "ExtCox002".Drv001.PowAct := "FC_NoiseReal"(Base := 19.6, Amp := #Amp_PowKw, Lo := #Lo, Hi := #Hi, Seed := #Seed);
	    "ExtCox002".Drv001.SpdSet := "FC_NoiseReal"(Base := 48.0, Amp := #Amp_SpdRpm, Lo := #Lo, Hi := #Hi, Seed := #Seed);
	    "ExtCox002".Drv001.SpdAct := "FC_NoiseReal"(Base := 48.0, Amp := #Amp_SpdRpm, Lo := #Lo, Hi := #Hi, Seed := #Seed);
	    "ExtCox002".Drv001.LoaAct := "FC_NoiseReal"(Base := 19.0, Amp := #Amp_LoaPct, Lo := #Lo, Hi := #Hi, Seed := #Seed);

	    // =========================
	    // Pressure & Melt Temp
	    // =========================
	    "ExtCox002".Prs001.Act := "FC_NoiseReal"(Base := 126.7, Amp := #Amp_PrsBar, Lo := #Lo, Hi := #Hi, Seed := #Seed); // Press P7
	    "ExtCox002".Prs002.Act := "FC_NoiseReal"(Base := 91.2, Amp := #Amp_PrsBar, Lo := #Lo, Hi := #Hi, Seed := #Seed); // Press P8
	    "ExtCox002".Prs012.Act := "FC_NoiseReal"(Base := 35.5, Amp := #Amp_PrsBar, Lo := #Lo, Hi := #Hi, Seed := #Seed); // Diff Press
	    "ExtCox002".TmpMel001.Act := "FC_NoiseReal"(Base := 258.5, Amp := #Amp_TmpC, Lo := #Lo, Hi := #Hi, Seed := #Seed); // Temp. Melt

	    // =========================
	    // All Zone (global setpoint)
	    // =========================
	    "ExtCox002".TmpAll.Set := "FC_NoiseReal"(Base := 267.0, Amp := #Amp_TmpC, Lo := #Lo, Hi := #Hi, Seed := #Seed);

	    // =========================
	    // Cylinder Zones 1..6
	    // =========================
	    // Zone 1
	    "ExtCox002".TmpCyl001.Set := "FC_NoiseReal"(Base := 267.0, Amp := #Amp_TmpC, Lo := #Lo, Hi := #Hi, Seed := #Seed);
	    "ExtCox002".TmpCyl001.Act := "FC_NoiseReal"(Base := 267.1, Amp := #Amp_TmpC, Lo := #Lo, Hi := #Hi, Seed := #Seed);
	    "ExtCox002".TmpCyl001.Y := "FC_NoiseReal"(Base := 82.0, Amp := #Amp_Y_Pct, Lo := #Lo, Hi := #Hi, Seed := #Seed);

	    // Zone 2
	    "ExtCox002".TmpCyl002.Set := "FC_NoiseReal"(Base := 267.0, Amp := #Amp_TmpC, Lo := #Lo, Hi := #Hi, Seed := #Seed);
	    "ExtCox002".TmpCyl002.Act := "FC_NoiseReal"(Base := 267.0, Amp := #Amp_TmpC, Lo := #Lo, Hi := #Hi, Seed := #Seed);
	    "ExtCox002".TmpCyl002.Y := "FC_NoiseReal"(Base := 49.0, Amp := #Amp_Y_Pct, Lo := #Lo, Hi := #Hi, Seed := #Seed);

	    // Zone 3
	    "ExtCox002".TmpCyl003.Set := "FC_NoiseReal"(Base := 267.0, Amp := #Amp_TmpC, Lo := #Lo, Hi := #Hi, Seed := #Seed);
	    "ExtCox002".TmpCyl003.Act := "FC_NoiseReal"(Base := 267.1, Amp := #Amp_TmpC, Lo := #Lo, Hi := #Hi, Seed := #Seed);
	    "ExtCox002".TmpCyl003.Y := "FC_NoiseReal"(Base := 47.0, Amp := #Amp_Y_Pct, Lo := #Lo, Hi := #Hi, Seed := #Seed);

	    // Zone 4
	    "ExtCox002".TmpCyl004.Set := "FC_NoiseReal"(Base := 265.0, Amp := #Amp_TmpC, Lo := #Lo, Hi := #Hi, Seed := #Seed);
	    "ExtCox002".TmpCyl004.Act := "FC_NoiseReal"(Base := 265.0, Amp := #Amp_TmpC, Lo := #Lo, Hi := #Hi, Seed := #Seed);
	    "ExtCox002".TmpCyl004.Y := "FC_NoiseReal"(Base := 31.0, Amp := #Amp_Y_Pct, Lo := #Lo, Hi := #Hi, Seed := #Seed);

	    // Zone 5
	    "ExtCox002".TmpCyl005.Set := "FC_NoiseReal"(Base := 265.0, Amp := #Amp_TmpC, Lo := #Lo, Hi := #Hi, Seed := #Seed);
	    "ExtCox002".TmpCyl005.Act := "FC_NoiseReal"(Base := 265.0, Amp := #Amp_TmpC, Lo := #Lo, Hi := #Hi, Seed := #Seed);
	    "ExtCox002".TmpCyl005.Y := "FC_NoiseReal"(Base := 12.0, Amp := #Amp_Y_Pct, Lo := #Lo, Hi := #Hi, Seed := #Seed);

	    // Zone 6
	    "ExtCox002".TmpCyl006.Set := "FC_NoiseReal"(Base := 265.0, Amp := #Amp_TmpC, Lo := #Lo, Hi := #Hi, Seed := #Seed);
	    "ExtCox002".TmpCyl006.Act := "FC_NoiseReal"(Base := 265.0, Amp := #Amp_TmpC, Lo := #Lo, Hi := #Hi, Seed := #Seed);
	    "ExtCox002".TmpCyl006.Y := "FC_NoiseReal"(Base := 9.0, Amp := #Amp_Y_Pct, Lo := #Lo, Hi := #Hi, Seed := #Seed);

	    // =========================
	    // Filter (kotak bawah tulisan "Filter": 265 / 264.1 / 59%)
	    // =========================
	    "ExtCox002".TmpFil.Set := "FC_NoiseReal"(Base := 265.0, Amp := #Amp_TmpC, Lo := #Lo, Hi := #Hi, Seed := #Seed);
	    "ExtCox002".TmpFil.Act := "FC_NoiseReal"(Base := 264.1, Amp := #Amp_TmpC, Lo := #Lo, Hi := #Hi, Seed := #Seed);
	    "ExtCox002".TmpFil.Y := "FC_NoiseReal"(Base := 59.0, Amp := #Amp_Y_Pct, Lo := #Lo, Hi := #Hi, Seed := #Seed);

	    // =========================
	    // Pipe 1 (265 / 264.1 / 59%)
	    // =========================
	    "ExtCox002".TmpPip001.Set := "FC_NoiseReal"(Base := 265.0, Amp := #Amp_TmpC, Lo := #Lo, Hi := #Hi, Seed := #Seed);
	    "ExtCox002".TmpPip001.Act := "FC_NoiseReal"(Base := 264.1, Amp := #Amp_TmpC, Lo := #Lo, Hi := #Hi, Seed := #Seed);
	    "ExtCox002".TmpPip001.Y := "FC_NoiseReal"(Base := 59.0, Amp := #Amp_Y_Pct, Lo := #Lo, Hi := #Hi, Seed := #Seed);

	    // =========================
	    // Pipe 2.1 .. 2.3
	    // =========================
	    "ExtCox002".TmpPip021.Set := "FC_NoiseReal"(Base := 265.0, Amp := #Amp_TmpC, Lo := #Lo, Hi := #Hi, Seed := #Seed);
	    "ExtCox002".TmpPip021.Act := "FC_NoiseReal"(Base := 264.3, Amp := #Amp_TmpC, Lo := #Lo, Hi := #Hi, Seed := #Seed);
	    "ExtCox002".TmpPip021.Y := "FC_NoiseReal"(Base := 83.0, Amp := #Amp_Y_Pct, Lo := #Lo, Hi := #Hi, Seed := #Seed);

	    "ExtCox002".TmpPip022.Set := "FC_NoiseReal"(Base := 265.0, Amp := #Amp_TmpC, Lo := #Lo, Hi := #Hi, Seed := #Seed);
	    "ExtCox002".TmpPip022.Act := "FC_NoiseReal"(Base := 265.0, Amp := #Amp_TmpC, Lo := #Lo, Hi := #Hi, Seed := #Seed);
	    "ExtCox002".TmpPip022.Y := "FC_NoiseReal"(Base := 23.0, Amp := #Amp_Y_Pct, Lo := #Lo, Hi := #Hi, Seed := #Seed);

	    "ExtCox002".TmpPip023.Set := "FC_NoiseReal"(Base := 265.0, Amp := #Amp_TmpC, Lo := #Lo, Hi := #Hi, Seed := #Seed);
	    "ExtCox002".TmpPip023.Act := "FC_NoiseReal"(Base := 265.0, Amp := #Amp_TmpC, Lo := #Lo, Hi := #Hi, Seed := #Seed);
	    "ExtCox002".TmpPip023.Y := "FC_NoiseReal"(Base := 23.0, Amp := #Amp_Y_Pct, Lo := #Lo, Hi := #Hi, Seed := #Seed);

	    // =========================
	    // TmpSch001 (kotak 100.0Â°C / 1999.9Â°C / 0.0%)
	    // =========================
	    "ExtCox002".TmpSch001.Set := "FC_NoiseReal"(Base := 100.0, Amp := #Amp_TmpC, Lo := #Lo, Hi := #Hi, Seed := #Seed);
	    "ExtCox002".TmpSch001.Act := "FC_NoiseReal"(Base := 1999.9, Amp := #Amp_TmpC, Lo := #Lo, Hi := #Hi, Seed := #Seed);
	    "ExtCox002".TmpSch001.Y := "FC_NoiseReal"(Base := 0.0, Amp := #Amp_Y_Pct, Lo := #Lo, Hi := #Hi, Seed := #Seed);

	    // TmpSch002 (tidak terlihat di gambar ini â†’ default sementara)
	    "ExtCox002".TmpSch002.Set := "FC_NoiseReal"(Base := 0.0, Amp := #Amp_TmpC, Lo := #Lo, Hi := #Hi, Seed := #Seed);
	    "ExtCox002".TmpSch002.Act := "FC_NoiseReal"(Base := 1999.9, Amp := #Amp_TmpC, Lo := #Lo, Hi := #Hi, Seed := #Seed);
	    "ExtCox002".TmpSch002.Y := "FC_NoiseReal"(Base := 0.0, Amp := #Amp_Y_Pct, Lo := #Lo, Hi := #Hi, Seed := #Seed);

END_FUNCTION

FUNCTION "FC_Fluct_DB311_ExtMel" : Void
{ S7_Optimized_Access := 'TRUE' }
VERSION : 0.1
// ============================================================
// FLUCTUATION DB311 (ExtMel)
// ============================================================
   VAR_INPUT
      Enable : Bool;   // amplitudo fluktuasi
      Amp_PowKw : Real;   // kW
      Amp_SpdRpm : Real;   // rpm
      Amp_TmpC : Real;   // degC
      Amp_PrsBar : Real;   // bar
      Amp_Y_Pct : Real;   // %
   END_VAR

   VAR_IN_OUT
      Seed : DInt;
   END_VAR

   VAR_TEMP
      Lo : Real;
      Hi : Real;
   END_VAR


BEGIN
	    IF NOT #Enable THEN
	        RETURN;
	    END_IF;

	    #Lo := -3.4E38;
	    #Hi := 3.4E38;

	    // ---- Drive ----
	    "ExtMel".Drv001.PowAct := "FC_NoiseReal"(Base := 0.0, Amp := #Amp_PowKw, Lo := #Lo, Hi := #Hi, Seed := #Seed);
	    "ExtMel".Drv001.SpdAct := "FC_NoiseReal"(Base := 132.9, Amp := #Amp_SpdRpm, Lo := #Lo, Hi := #Hi, Seed := #Seed);
	    "ExtMel".Drv001.SpdSet := "FC_NoiseReal"(Base := 132.9, Amp := #Amp_SpdRpm, Lo := #Lo, Hi := #Hi, Seed := #Seed);
	    "ExtMel".Drv001.TmpAct := "FC_NoiseReal"(Base := 60.0, Amp := #Amp_TmpC, Lo := #Lo, Hi := #Hi, Seed := #Seed);
	    "ExtMel".Drv001.LoaAct := "FC_NoiseReal"(Base := 63.1, Amp := #Amp_PrsBar, Lo := #Lo, Hi := #Hi, Seed := #Seed);

	    // ---- Melt temperature ----
	    "ExtMel".TmpMel001.Act := "FC_NoiseReal"(Base := 208.0, Amp := #Amp_TmpC, Lo := #Lo, Hi := #Hi, Seed := #Seed);

	    // ---- Pressure ----
	    "ExtMel".Prs001.Act := "FC_NoiseReal"(Base := 34.8, Amp := #Amp_PrsBar, Lo := #Lo, Hi := #Hi, Seed := #Seed);
	    "ExtMel".PrsCtl.Act := "FC_NoiseReal"(Base := 34.2, Amp := #Amp_PrsBar, Lo := #Lo, Hi := #Hi, Seed := #Seed);
	    "ExtMel".PrsCtl.Set := "FC_NoiseReal"(Base := 35.0, Amp := #Amp_PrsBar, Lo := #Lo, Hi := #Hi, Seed := #Seed);
	    "ExtMel".PrsCtl.Y := "FC_NoiseReal"(Base := 44.6, Amp := #Amp_Y_Pct, Lo := #Lo, Hi := #Hi, Seed := #Seed);
	    "ExtMel".PmtPrsCtl.Y := "FC_NoiseReal"(Base := 44.6, Amp := #Amp_Y_Pct, Lo := #Lo, Hi := #Hi, Seed := #Seed);

	    // ---- All Zone setpoint ----
	    "ExtMel".TmpAll.Set := "FC_NoiseReal"(Base := 235.0, Amp := #Amp_TmpC, Lo := #Lo, Hi := #Hi, Seed := #Seed);

	    // ---- Feeding ----
	    "ExtMel".TmpFdg.Act := "FC_NoiseReal"(Base := 31.8, Amp := #Amp_TmpC, Lo := #Lo, Hi := #Hi, Seed := #Seed);
	    "ExtMel".TmpFdg.Set := "FC_NoiseReal"(Base := 32.0, Amp := #Amp_TmpC, Lo := #Lo, Hi := #Hi, Seed := #Seed);
	    "ExtMel".TmpFdg.Y := "FC_NoiseReal"(Base := -15.0, Amp := #Amp_Y_Pct, Lo := #Lo, Hi := #Hi, Seed := #Seed);

	    // ---- Zone 1 ----
	    "ExtMel".TmpCyl001.Act := "FC_NoiseReal"(Base := 219.3, Amp := #Amp_TmpC, Lo := #Lo, Hi := #Hi, Seed := #Seed);
	    "ExtMel".TmpCyl001.Set := "FC_NoiseReal"(Base := 220.0, Amp := #Amp_TmpC, Lo := #Lo, Hi := #Hi, Seed := #Seed);
	    "ExtMel".TmpCyl001.Y := "FC_NoiseReal"(Base := 51.0, Amp := #Amp_Y_Pct, Lo := #Lo, Hi := #Hi, Seed := #Seed);

	    // ---- Zone 2 ----
	    "ExtMel".TmpCyl002.Act := "FC_NoiseReal"(Base := 228.6, Amp := #Amp_TmpC, Lo := #Lo, Hi := #Hi, Seed := #Seed);
	    "ExtMel".TmpCyl002.Set := "FC_NoiseReal"(Base := 230.0, Amp := #Amp_TmpC, Lo := #Lo, Hi := #Hi, Seed := #Seed);
	    "ExtMel".TmpCyl002.Y := "FC_NoiseReal"(Base := 11.0, Amp := #Amp_Y_Pct, Lo := #Lo, Hi := #Hi, Seed := #Seed);

	    // ---- Zone 3 ----
	    "ExtMel".TmpCyl003.Act := "FC_NoiseReal"(Base := 243.8, Amp := #Amp_TmpC, Lo := #Lo, Hi := #Hi, Seed := #Seed);
	    "ExtMel".TmpCyl003.Set := "FC_NoiseReal"(Base := 245.0, Amp := #Amp_TmpC, Lo := #Lo, Hi := #Hi, Seed := #Seed);
	    "ExtMel".TmpCyl003.Y := "FC_NoiseReal"(Base := 3.0, Amp := #Amp_Y_Pct, Lo := #Lo, Hi := #Hi, Seed := #Seed);

	    // ---- Zone 4 ----
	    "ExtMel".TmpCyl004.Act := "FC_NoiseReal"(Base := 240.2, Amp := #Amp_TmpC, Lo := #Lo, Hi := #Hi, Seed := #Seed);
	    "ExtMel".TmpCyl004.Set := "FC_NoiseReal"(Base := 240.0, Amp := #Amp_TmpC, Lo := #Lo, Hi := #Hi, Seed := #Seed);
	    "ExtMel".TmpCyl004.Y := "FC_NoiseReal"(Base := 0.0, Amp := #Amp_Y_Pct, Lo := #Lo, Hi := #Hi, Seed := #Seed);

	    // ---- Zone 5 ----
	    "ExtMel".TmpCyl005.Act := "FC_NoiseReal"(Base := 234.9, Amp := #Amp_TmpC, Lo := #Lo, Hi := #Hi, Seed := #Seed);
	    "ExtMel".TmpCyl005.Set := "FC_NoiseReal"(Base := 235.0, Amp := #Amp_TmpC, Lo := #Lo, Hi := #Hi, Seed := #Seed);
	    "ExtMel".TmpCyl005.Y := "FC_NoiseReal"(Base := 17.0, Amp := #Amp_Y_Pct, Lo := #Lo, Hi := #Hi, Seed := #Seed);

	    // ---- Zone 6 ----
	    "ExtMel".TmpCyl006.Act := "FC_NoiseReal"(Base := 234.3, Amp := #Amp_TmpC, Lo := #Lo, Hi := #Hi, Seed := #Seed);
	    "ExtMel".TmpCyl006.Set := "FC_NoiseReal"(Base := 235.0, Amp := #Amp_TmpC, Lo := #Lo, Hi := #Hi, Seed := #Seed);
	    "ExtMel".TmpCyl006.Y := "FC_NoiseReal"(Base := 11.0, Amp := #Amp_Y_Pct, Lo := #Lo, Hi := #Hi, Seed := #Seed);

	    // ---- Flange ----
	    "ExtMel".TmpFlg.Act := "FC_NoiseReal"(Base := 235.0, Amp := #Amp_TmpC, Lo := #Lo, Hi := #Hi, Seed := #Seed);
	    "ExtMel".TmpFlg.Set := "FC_NoiseReal"(Base := 235.0, Amp := #Amp_TmpC, Lo := #Lo, Hi := #Hi, Seed := #Seed);
	    "ExtMel".TmpFlg.Y := "FC_NoiseReal"(Base := 15.0, Amp := #Amp_Y_Pct, Lo := #Lo, Hi := #Hi, Seed := #Seed);

	    // ---- Adapter ----
	    "ExtMel".TmpAdp.Act := "FC_NoiseReal"(Base := 235.0, Amp := #Amp_TmpC, Lo := #Lo, Hi := #Hi, Seed := #Seed);
	    "ExtMel".TmpAdp.Set := "FC_NoiseReal"(Base := 235.0, Amp := #Amp_TmpC, Lo := #Lo, Hi := #Hi, Seed := #Seed);
	    "ExtMel".TmpAdp.Y := "FC_NoiseReal"(Base := 45.0, Amp := #Amp_Y_Pct, Lo := #Lo, Hi := #Hi, Seed := #Seed);

	    // ---- Melt Pipe ----
	    "ExtMel".TmpPip001.Act := "FC_NoiseReal"(Base := 235.0, Amp := #Amp_TmpC, Lo := #Lo, Hi := #Hi, Seed := #Seed);
	    "ExtMel".TmpPip001.Set := "FC_NoiseReal"(Base := 235.0, Amp := #Amp_TmpC, Lo := #Lo, Hi := #Hi, Seed := #Seed);
	    "ExtMel".TmpPip001.Y := "FC_NoiseReal"(Base := 17.0, Amp := #Amp_Y_Pct, Lo := #Lo, Hi := #Hi, Seed := #Seed);
END_FUNCTION

FUNCTION "FC_Fluct_DB316_ExtCox001" : Void
{ S7_Optimized_Access := 'TRUE' }
VERSION : 0.1
// ============================================================
// FLUCTUATION DB316 (ExtCox001)
// ============================================================
   VAR_INPUT
      Enable : Bool;   // amplitudo fluktuasi
      Amp_PowKw : Real;   // Â±kW
      Amp_SpdRpm : Real;   // Â±rpm
      Amp_LoaPct : Real;   // Â±%
      Amp_TmpC : Real;   // Â±Â°C
      Amp_PrsBar : Real;   // Â±bar
      Amp_Y_Pct : Real;   // Â±%
   END_VAR

   VAR_IN_OUT
      Seed : DInt;
   END_VAR

   VAR_TEMP
      Lo : Real;
      Hi : Real;
   END_VAR


BEGIN
	    IF NOT #Enable THEN
	        RETURN;
	    END_IF;

	    #Lo := -3.4E38;
	    #Hi := 3.4E38;

	    // =========================
	    // Drive (panel kiri bawah)
	    // =========================
	    "ExtCox001".Drv001.TmpAct := "FC_NoiseReal"(Base := 56.3, Amp := #Amp_TmpC, Lo := #Lo, Hi := #Hi, Seed := #Seed);
	    "ExtCox001".Drv001.PowAct := "FC_NoiseReal"(Base := 5.5, Amp := #Amp_PowKw, Lo := #Lo, Hi := #Hi, Seed := #Seed);
	    "ExtCox001".Drv001.SpdSet := "FC_NoiseReal"(Base := 23.0, Amp := #Amp_SpdRpm, Lo := #Lo, Hi := #Hi, Seed := #Seed);
	    "ExtCox001".Drv001.SpdAct := "FC_NoiseReal"(Base := 23.0, Amp := #Amp_SpdRpm, Lo := #Lo, Hi := #Hi, Seed := #Seed);
	    "ExtCox001".Drv001.LoaAct := "FC_NoiseReal"(Base := 11.1, Amp := #Amp_LoaPct, Lo := #Lo, Hi := #Hi, Seed := #Seed);

	    // =========================
	    // Pressure & Melt Temp
	    // =========================
	    "ExtCox001".Prs001.Act := "FC_NoiseReal"(Base := 105.1, Amp := #Amp_PrsBar, Lo := #Lo, Hi := #Hi, Seed := #Seed); // Press P5
	    "ExtCox001".Prs002.Act := "FC_NoiseReal"(Base := 58.8, Amp := #Amp_PrsBar, Lo := #Lo, Hi := #Hi, Seed := #Seed); // Press P6
	    "ExtCox001".Prs012.Act := "FC_NoiseReal"(Base := 46.3, Amp := #Amp_PrsBar, Lo := #Lo, Hi := #Hi, Seed := #Seed); // Diff Press
	    "ExtCox001".TmpMel001.Act := "FC_NoiseReal"(Base := 248.7, Amp := #Amp_TmpC, Lo := #Lo, Hi := #Hi, Seed := #Seed); // Temp. Melt

	    // =========================
	    // All Zone (global setpoint)
	    // =========================
	    "ExtCox001".TmpAll.Set := "FC_NoiseReal"(Base := 260.0, Amp := #Amp_TmpC, Lo := #Lo, Hi := #Hi, Seed := #Seed);

	    // =========================
	    // Cylinder Zones 1..6
	    // =========================
	    // Zone 1
	    "ExtCox001".TmpCyl001.Set := "FC_NoiseReal"(Base := 260.0, Amp := #Amp_TmpC, Lo := #Lo, Hi := #Hi, Seed := #Seed);
	    "ExtCox001".TmpCyl001.Act := "FC_NoiseReal"(Base := 260.2, Amp := #Amp_TmpC, Lo := #Lo, Hi := #Hi, Seed := #Seed);
	    "ExtCox001".TmpCyl001.Y := "FC_NoiseReal"(Base := 86.0, Amp := #Amp_Y_Pct, Lo := #Lo, Hi := #Hi, Seed := #Seed);

	    // Zone 2
	    "ExtCox001".TmpCyl002.Set := "FC_NoiseReal"(Base := 260.0, Amp := #Amp_TmpC, Lo := #Lo, Hi := #Hi, Seed := #Seed);
	    "ExtCox001".TmpCyl002.Act := "FC_NoiseReal"(Base := 260.0, Amp := #Amp_TmpC, Lo := #Lo, Hi := #Hi, Seed := #Seed);
	    "ExtCox001".TmpCyl002.Y := "FC_NoiseReal"(Base := 33.0, Amp := #Amp_Y_Pct, Lo := #Lo, Hi := #Hi, Seed := #Seed);

	    // Zone 3
	    "ExtCox001".TmpCyl003.Set := "FC_NoiseReal"(Base := 260.0, Amp := #Amp_TmpC, Lo := #Lo, Hi := #Hi, Seed := #Seed);
	    "ExtCox001".TmpCyl003.Act := "FC_NoiseReal"(Base := 260.1, Amp := #Amp_TmpC, Lo := #Lo, Hi := #Hi, Seed := #Seed);
	    "ExtCox001".TmpCyl003.Y := "FC_NoiseReal"(Base := 24.0, Amp := #Amp_Y_Pct, Lo := #Lo, Hi := #Hi, Seed := #Seed);

	    // Zone 4
	    "ExtCox001".TmpCyl004.Set := "FC_NoiseReal"(Base := 255.0, Amp := #Amp_TmpC, Lo := #Lo, Hi := #Hi, Seed := #Seed);
	    "ExtCox001".TmpCyl004.Act := "FC_NoiseReal"(Base := 255.0, Amp := #Amp_TmpC, Lo := #Lo, Hi := #Hi, Seed := #Seed);
	    "ExtCox001".TmpCyl004.Y := "FC_NoiseReal"(Base := 10.0, Amp := #Amp_Y_Pct, Lo := #Lo, Hi := #Hi, Seed := #Seed);

	    // Zone 5
	    "ExtCox001".TmpCyl005.Set := "FC_NoiseReal"(Base := 255.0, Amp := #Amp_TmpC, Lo := #Lo, Hi := #Hi, Seed := #Seed);
	    "ExtCox001".TmpCyl005.Act := "FC_NoiseReal"(Base := 255.3, Amp := #Amp_TmpC, Lo := #Lo, Hi := #Hi, Seed := #Seed);
	    "ExtCox001".TmpCyl005.Y := "FC_NoiseReal"(Base := 0.0, Amp := #Amp_Y_Pct, Lo := #Lo, Hi := #Hi, Seed := #Seed);

	    // Zone 6
	    "ExtCox001".TmpCyl006.Set := "FC_NoiseReal"(Base := 255.0, Amp := #Amp_TmpC, Lo := #Lo, Hi := #Hi, Seed := #Seed);
	    "ExtCox001".TmpCyl006.Act := "FC_NoiseReal"(Base := 255.1, Amp := #Amp_TmpC, Lo := #Lo, Hi := #Hi, Seed := #Seed);
	    "ExtCox001".TmpCyl006.Y := "FC_NoiseReal"(Base := 21.0, Amp := #Amp_Y_Pct, Lo := #Lo, Hi := #Hi, Seed := #Seed);

	    // =========================
	    // Filter (kotak di bawah tulisan "Filter": 255/255/35%)
	    // =========================
	    "ExtCox001".TmpFil.Set := "FC_NoiseReal"(Base := 255.0, Amp := #Amp_TmpC, Lo := #Lo, Hi := #Hi, Seed := #Seed);
	    "ExtCox001".TmpFil.Act := "FC_NoiseReal"(Base := 255.0, Amp := #Amp_TmpC, Lo := #Lo, Hi := #Hi, Seed := #Seed);
	    "ExtCox001".TmpFil.Y := "FC_NoiseReal"(Base := 35.0, Amp := #Amp_Y_Pct, Lo := #Lo, Hi := #Hi, Seed := #Seed);

	    // =========================
	    // Pipe 1 (255/255/45%)
	    // =========================
	    "ExtCox001".TmpPip001.Set := "FC_NoiseReal"(Base := 255.0, Amp := #Amp_TmpC, Lo := #Lo, Hi := #Hi, Seed := #Seed);
	    "ExtCox001".TmpPip001.Act := "FC_NoiseReal"(Base := 255.0, Amp := #Amp_TmpC, Lo := #Lo, Hi := #Hi, Seed := #Seed);
	    "ExtCox001".TmpPip001.Y := "FC_NoiseReal"(Base := 45.0, Amp := #Amp_Y_Pct, Lo := #Lo, Hi := #Hi, Seed := #Seed);

	    // =========================
	    // Pipe 2.1 .. 2.3
	    // =========================
	    "ExtCox001".TmpPip021.Set := "FC_NoiseReal"(Base := 255.0, Amp := #Amp_TmpC, Lo := #Lo, Hi := #Hi, Seed := #Seed);
	    "ExtCox001".TmpPip021.Act := "FC_NoiseReal"(Base := 255.0, Amp := #Amp_TmpC, Lo := #Lo, Hi := #Hi, Seed := #Seed);
	    "ExtCox001".TmpPip021.Y := "FC_NoiseReal"(Base := 42.0, Amp := #Amp_Y_Pct, Lo := #Lo, Hi := #Hi, Seed := #Seed);

	    "ExtCox001".TmpPip022.Set := "FC_NoiseReal"(Base := 255.0, Amp := #Amp_TmpC, Lo := #Lo, Hi := #Hi, Seed := #Seed);
	    "ExtCox001".TmpPip022.Act := "FC_NoiseReal"(Base := 254.4, Amp := #Amp_TmpC, Lo := #Lo, Hi := #Hi, Seed := #Seed);
	    "ExtCox001".TmpPip022.Y := "FC_NoiseReal"(Base := 37.0, Amp := #Amp_Y_Pct, Lo := #Lo, Hi := #Hi, Seed := #Seed);

	    "ExtCox001".TmpPip023.Set := "FC_NoiseReal"(Base := 255.0, Amp := #Amp_TmpC, Lo := #Lo, Hi := #Hi, Seed := #Seed);
	    "ExtCox001".TmpPip023.Act := "FC_NoiseReal"(Base := 253.2, Amp := #Amp_TmpC, Lo := #Lo, Hi := #Hi, Seed := #Seed);
	    "ExtCox001".TmpPip023.Y := "FC_NoiseReal"(Base := 47.0, Amp := #Amp_Y_Pct, Lo := #Lo, Hi := #Hi, Seed := #Seed);

	    // =========================
	    // "TmpSch" (kotak 70.0Â°C / 1999.9Â°C / 0.0% di gambar)
	    // =========================
	    "ExtCox001".TmpSch001.Set := "FC_NoiseReal"(Base := 255.0, Amp := #Amp_TmpC, Lo := #Lo, Hi := #Hi, Seed := #Seed);
	    "ExtCox001".TmpSch001.Act := "FC_NoiseReal"(Base := 255.0, Amp := #Amp_TmpC, Lo := #Lo, Hi := #Hi, Seed := #Seed);
	    "ExtCox001".TmpSch001.Y := "FC_NoiseReal"(Base := 33.0, Amp := #Amp_Y_Pct, Lo := #Lo, Hi := #Hi, Seed := #Seed);

	    // TmpSch002 (tidak terlihat di gambar ini â†’ default sementara)
	    "ExtCox001".TmpSch002.Set := "FC_NoiseReal"(Base := 70.0, Amp := #Amp_TmpC, Lo := #Lo, Hi := #Hi, Seed := #Seed);
	    "ExtCox001".TmpSch002.Act := "FC_NoiseReal"(Base := 70.0, Amp := #Amp_TmpC, Lo := #Lo, Hi := #Hi, Seed := #Seed);
	    "ExtCox001".TmpSch002.Y := "FC_NoiseReal"(Base := 0.0, Amp := #Amp_Y_Pct, Lo := #Lo, Hi := #Hi, Seed := #Seed);

END_FUNCTION

FUNCTION "FC_Fluct_DB315_ExtDieBlt" : Void
{ S7_Optimized_Access := 'TRUE' }
VERSION : 0.1
// ============================================================
// FLUCTUATION DB315 (ExtDieBlt)
// ============================================================
   VAR_INPUT
      Enable : Bool;
      Amp_TmpC : Real;   // Â±Â°C
   END_VAR

   VAR_IN_OUT
      Seed : DInt;
   END_VAR

   VAR_TEMP
      Lo : Real;
      Hi : Real;
   END_VAR


BEGIN
	    IF NOT #Enable THEN
	        RETURN;
	    END_IF;

	    #Lo := -3.4E38;
	    #Hi := 3.4E38;

	    // ---- Bolt 1..10 ----
	    "ExtDieBlt".TmpBlt[1].Act := "FC_NoiseReal"(Base := 208.3, Amp := #Amp_TmpC, Lo := #Lo, Hi := #Hi, Seed := #Seed);
	    "ExtDieBlt".TmpBlt[2].Act := "FC_NoiseReal"(Base := 233.1, Amp := #Amp_TmpC, Lo := #Lo, Hi := #Hi, Seed := #Seed);
	    "ExtDieBlt".TmpBlt[3].Act := "FC_NoiseReal"(Base := 220.5, Amp := #Amp_TmpC, Lo := #Lo, Hi := #Hi, Seed := #Seed);
	    "ExtDieBlt".TmpBlt[4].Act := "FC_NoiseReal"(Base := 209.2, Amp := #Amp_TmpC, Lo := #Lo, Hi := #Hi, Seed := #Seed);
	    "ExtDieBlt".TmpBlt[5].Act := "FC_NoiseReal"(Base := 227.0, Amp := #Amp_TmpC, Lo := #Lo, Hi := #Hi, Seed := #Seed);
	    "ExtDieBlt".TmpBlt[6].Act := "FC_NoiseReal"(Base := 222.0, Amp := #Amp_TmpC, Lo := #Lo, Hi := #Hi, Seed := #Seed);
	    "ExtDieBlt".TmpBlt[7].Act := "FC_NoiseReal"(Base := 223.8, Amp := #Amp_TmpC, Lo := #Lo, Hi := #Hi, Seed := #Seed);
	    "ExtDieBlt".TmpBlt[08].Act := "FC_NoiseReal"(Base := 180.4, Amp := #Amp_TmpC, Lo := #Lo, Hi := #Hi, Seed := #Seed);
	    "ExtDieBlt".TmpBlt[09].Act := "FC_NoiseReal"(Base := 225.2, Amp := #Amp_TmpC, Lo := #Lo, Hi := #Hi, Seed := #Seed);
	    "ExtDieBlt".TmpBlt[10].Act := "FC_NoiseReal"(Base := 196.3, Amp := #Amp_TmpC, Lo := #Lo, Hi := #Hi, Seed := #Seed);

	    // ---- Bolt 11..20 ----
	    "ExtDieBlt".TmpBlt[11].Act := "FC_NoiseReal"(Base := 231.1, Amp := #Amp_TmpC, Lo := #Lo, Hi := #Hi, Seed := #Seed);
	    "ExtDieBlt".TmpBlt[12].Act := "FC_NoiseReal"(Base := 228.5, Amp := #Amp_TmpC, Lo := #Lo, Hi := #Hi, Seed := #Seed);
	    "ExtDieBlt".TmpBlt[13].Act := "FC_NoiseReal"(Base := 235.6, Amp := #Amp_TmpC, Lo := #Lo, Hi := #Hi, Seed := #Seed);
	    "ExtDieBlt".TmpBlt[14].Act := "FC_NoiseReal"(Base := 215.6, Amp := #Amp_TmpC, Lo := #Lo, Hi := #Hi, Seed := #Seed);
	    "ExtDieBlt".TmpBlt[15].Act := "FC_NoiseReal"(Base := 215.5, Amp := #Amp_TmpC, Lo := #Lo, Hi := #Hi, Seed := #Seed);
	    "ExtDieBlt".TmpBlt[16].Act := "FC_NoiseReal"(Base := 213.0, Amp := #Amp_TmpC, Lo := #Lo, Hi := #Hi, Seed := #Seed);
	    "ExtDieBlt".TmpBlt[17].Act := "FC_NoiseReal"(Base := 200.8, Amp := #Amp_TmpC, Lo := #Lo, Hi := #Hi, Seed := #Seed);
	    "ExtDieBlt".TmpBlt[18].Act := "FC_NoiseReal"(Base := 228.4, Amp := #Amp_TmpC, Lo := #Lo, Hi := #Hi, Seed := #Seed);
	    "ExtDieBlt".TmpBlt[19].Act := "FC_NoiseReal"(Base := 195.8, Amp := #Amp_TmpC, Lo := #Lo, Hi := #Hi, Seed := #Seed);
	    "ExtDieBlt".TmpBlt[20].Act := "FC_NoiseReal"(Base := 212.0, Amp := #Amp_TmpC, Lo := #Lo, Hi := #Hi, Seed := #Seed);

	    // ---- Bolt 21..30 ----
	    "ExtDieBlt".TmpBlt[21].Act := "FC_NoiseReal"(Base := 214.7, Amp := #Amp_TmpC, Lo := #Lo, Hi := #Hi, Seed := #Seed);
	    "ExtDieBlt".TmpBlt[22].Act := "FC_NoiseReal"(Base := 217.3, Amp := #Amp_TmpC, Lo := #Lo, Hi := #Hi, Seed := #Seed);
	    "ExtDieBlt".TmpBlt[23].Act := "FC_NoiseReal"(Base := 229.2, Amp := #Amp_TmpC, Lo := #Lo, Hi := #Hi, Seed := #Seed);
	    "ExtDieBlt".TmpBlt[24].Act := "FC_NoiseReal"(Base := 231.2, Amp := #Amp_TmpC, Lo := #Lo, Hi := #Hi, Seed := #Seed);
	    "ExtDieBlt".TmpBlt[25].Act := "FC_NoiseReal"(Base := 220.0, Amp := #Amp_TmpC, Lo := #Lo, Hi := #Hi, Seed := #Seed);
	    "ExtDieBlt".TmpBlt[26].Act := "FC_NoiseReal"(Base := 226.0, Amp := #Amp_TmpC, Lo := #Lo, Hi := #Hi, Seed := #Seed);
	    "ExtDieBlt".TmpBlt[27].Act := "FC_NoiseReal"(Base := 219.6, Amp := #Amp_TmpC, Lo := #Lo, Hi := #Hi, Seed := #Seed);
	    "ExtDieBlt".TmpBlt[28].Act := "FC_NoiseReal"(Base := 219.2, Amp := #Amp_TmpC, Lo := #Lo, Hi := #Hi, Seed := #Seed);
	    "ExtDieBlt".TmpBlt[29].Act := "FC_NoiseReal"(Base := 226.4, Amp := #Amp_TmpC, Lo := #Lo, Hi := #Hi, Seed := #Seed);
	    "ExtDieBlt".TmpBlt[30].Act := "FC_NoiseReal"(Base := 212.5, Amp := #Amp_TmpC, Lo := #Lo, Hi := #Hi, Seed := #Seed);

	    // ---- Bolt 31 (tidak terlihat di gambar yang kamu kirim) ----
	    "ExtDieBlt".TmpBlt[31].Act := 560;

END_FUNCTION

FUNCTION "FC_Fluct_DB312_ExtMet" : Void
{ S7_Optimized_Access := 'TRUE' }
VERSION : 0.1
// ============================================================
// FLUCTUATION AREA: DB312 / "ExtMet"
// ============================================================
   VAR_INPUT
      Enable : Bool;
      Amp_PowKw : Real;   // Â±kW
      Amp_SpdRpm : Real;   // Â±rpm
      Amp_TmpC : Real;   // Â±Â°C
      Amp_Y_Pct : Real;   // Â±%
      Amp_PrsBar : Real;   // Â±bar
   END_VAR

   VAR_IN_OUT
      Seed : DInt;
   END_VAR

   VAR_TEMP
      Lo : Real;
      Hi : Real;
   END_VAR


BEGIN
	    IF NOT #Enable THEN
	        RETURN;
	    END_IF;

	    #Lo := -3.4E38;
	    #Hi := 3.4E38;

	    // ---- Drive ----
	    "ExtMet".Drv001.PowAct := "FC_NoiseReal"(Base := 157.4, Amp := #Amp_PowKw, Lo := #Lo, Hi := #Hi, Seed := #Seed);
	    "ExtMet".Drv001.SpdAct := "FC_NoiseReal"(Base := 54.5, Amp := #Amp_SpdRpm, Lo := #Lo, Hi := #Hi, Seed := #Seed);
	    "ExtMet".Drv001.SpdSet := "FC_NoiseReal"(Base := 54.5, Amp := #Amp_SpdRpm, Lo := #Lo, Hi := #Hi, Seed := #Seed);
	    "ExtMet".Drv001.TmpAct := "FC_NoiseReal"(Base := 69.1, Amp := #Amp_TmpC, Lo := #Lo, Hi := #Hi, Seed := #Seed);
	    "ExtMet".Drv001.LoaAct := "FC_NoiseReal"(Base := 65.8, Amp := #Amp_PrsBar, Lo := #Lo, Hi := #Hi, Seed := #Seed);

	    // ---- All Zone ----
	    "ExtMet".TmpAll.Set := "FC_NoiseReal"(Base := 235.0, Amp := #Amp_TmpC, Lo := #Lo, Hi := #Hi, Seed := #Seed);

	    // ---- Zone 1 ----
	    "ExtMet".TmpCyl001.Act := "FC_NoiseReal"(Base := 235.2, Amp := #Amp_TmpC, Lo := #Lo, Hi := #Hi, Seed := #Seed);
	    "ExtMet".TmpCyl001.Set := "FC_NoiseReal"(Base := 235.0, Amp := #Amp_TmpC, Lo := #Lo, Hi := #Hi, Seed := #Seed);
	    "ExtMet".TmpCyl001.Y := "FC_NoiseReal"(Base := 55.0, Amp := #Amp_Y_Pct, Lo := #Lo, Hi := #Hi, Seed := #Seed);

	    // ---- Zone 2 ----
	    "ExtMet".TmpCyl002.Act := "FC_NoiseReal"(Base := 235.5, Amp := #Amp_TmpC, Lo := #Lo, Hi := #Hi, Seed := #Seed);
	    "ExtMet".TmpCyl002.Set := "FC_NoiseReal"(Base := 235.0, Amp := #Amp_TmpC, Lo := #Lo, Hi := #Hi, Seed := #Seed);
	    "ExtMet".TmpCyl002.Y := "FC_NoiseReal"(Base := 0.0, Amp := #Amp_Y_Pct, Lo := #Lo, Hi := #Hi, Seed := #Seed);

	    // ---- Zone 3 ----
	    "ExtMet".TmpCyl003.Act := "FC_NoiseReal"(Base := 235.3, Amp := #Amp_TmpC, Lo := #Lo, Hi := #Hi, Seed := #Seed);
	    "ExtMet".TmpCyl003.Set := "FC_NoiseReal"(Base := 235.0, Amp := #Amp_TmpC, Lo := #Lo, Hi := #Hi, Seed := #Seed);
	    "ExtMet".TmpCyl003.Y := "FC_NoiseReal"(Base := -3.0, Amp := #Amp_Y_Pct, Lo := #Lo, Hi := #Hi, Seed := #Seed);

	    // ---- Zone 4 ----
	    "ExtMet".TmpCyl004.Act := "FC_NoiseReal"(Base := 234.8, Amp := #Amp_TmpC, Lo := #Lo, Hi := #Hi, Seed := #Seed);
	    "ExtMet".TmpCyl004.Set := "FC_NoiseReal"(Base := 235.0, Amp := #Amp_TmpC, Lo := #Lo, Hi := #Hi, Seed := #Seed);
	    "ExtMet".TmpCyl004.Y := "FC_NoiseReal"(Base := 0.0, Amp := #Amp_Y_Pct, Lo := #Lo, Hi := #Hi, Seed := #Seed);

	    // ---- Zone 5 ----
	    "ExtMet".TmpCyl005.Act := "FC_NoiseReal"(Base := 235.7, Amp := #Amp_TmpC, Lo := #Lo, Hi := #Hi, Seed := #Seed);
	    "ExtMet".TmpCyl005.Set := "FC_NoiseReal"(Base := 235.0, Amp := #Amp_TmpC, Lo := #Lo, Hi := #Hi, Seed := #Seed);
	    "ExtMet".TmpCyl005.Y := "FC_NoiseReal"(Base := -4.0, Amp := #Amp_Y_Pct, Lo := #Lo, Hi := #Hi, Seed := #Seed);

	    // ---- Zone 6 ----
	    "ExtMet".TmpCyl006.Act := "FC_NoiseReal"(Base := 235.1, Amp := #Amp_TmpC, Lo := #Lo, Hi := #Hi, Seed := #Seed);
	    "ExtMet".TmpCyl006.Set := "FC_NoiseReal"(Base := 235.0, Amp := #Amp_TmpC, Lo := #Lo, Hi := #Hi, Seed := #Seed);
	    "ExtMet".TmpCyl006.Y := "FC_NoiseReal"(Base := -3.0, Amp := #Amp_Y_Pct, Lo := #Lo, Hi := #Hi, Seed := #Seed);

	    // ---- Zone 7 ----
	    "ExtMet".TmpCyl007.Act := "FC_NoiseReal"(Base := 235.0, Amp := #Amp_TmpC, Lo := #Lo, Hi := #Hi, Seed := #Seed);
	    "ExtMet".TmpCyl007.Set := "FC_NoiseReal"(Base := 235.0, Amp := #Amp_TmpC, Lo := #Lo, Hi := #Hi, Seed := #Seed);
	    "ExtMet".TmpCyl007.Y := "FC_NoiseReal"(Base := -1.0, Amp := #Amp_Y_Pct, Lo := #Lo, Hi := #Hi, Seed := #Seed);

	    // ---- Flange ----
	    "ExtMet".TmpFlg.Act := "FC_NoiseReal"(Base := 235.1, Amp := #Amp_TmpC, Lo := #Lo, Hi := #Hi, Seed := #Seed);
	    "ExtMet".TmpFlg.Set := "FC_NoiseReal"(Base := 235.0, Amp := #Amp_TmpC, Lo := #Lo, Hi := #Hi, Seed := #Seed);
	    "ExtMet".TmpFlg.Y := "FC_NoiseReal"(Base := 33.0, Amp := #Amp_Y_Pct, Lo := #Lo, Hi := #Hi, Seed := #Seed);

END_FUNCTION

FUNCTION "FC_Fluct_DB314_ExtDie" : Void
{ S7_Optimized_Access := 'TRUE' }
VERSION : 0.1
// ============================================================
// FLUCTUATION DB314 (ExtDie)
// ============================================================
   VAR_INPUT
      Enable : Bool;   // amplitudo fluktuasi
      Amp_TmpC : Real;   // Â±Â°C
      Amp_Y_Pct : Real;   // Â±%
   END_VAR

   VAR_IN_OUT
      Seed : DInt;
   END_VAR

   VAR_TEMP
      Lo : Real;
      Hi : Real;
   END_VAR


BEGIN
	    IF NOT #Enable THEN
	        RETURN;
	    END_IF;

	    #Lo := -3.4E38;
	    #Hi := 3.4E38;

	    // =========================
	    // All Zone
	    // =========================
	    "ExtDie".TmpAll.Set := "FC_NoiseReal"(Base := 250.0, Amp := #Amp_TmpC, Lo := #Lo, Hi := #Hi, Seed := #Seed);

	    // =========================
	    // Adapter 1
	    // (Set 250.0 / Act 250.2 / Y 33.0)
	    // =========================
	    "ExtDie".TmpAdp001.Set := "FC_NoiseReal"(Base := 250.0, Amp := #Amp_TmpC, Lo := #Lo, Hi := #Hi, Seed := #Seed);
	    "ExtDie".TmpAdp001.Act := "FC_NoiseReal"(Base := 250.2, Amp := #Amp_TmpC, Lo := #Lo, Hi := #Hi, Seed := #Seed);
	    "ExtDie".TmpAdp001.Y := "FC_NoiseReal"(Base := 33.0, Amp := #Amp_Y_Pct, Lo := #Lo, Hi := #Hi, Seed := #Seed);

	    // =========================
	    // Adapter 2
	    // (Set 250.0 / Act 249.9 / Y 45.0)
	    // =========================
	    "ExtDie".TmpAdp002.Set := "FC_NoiseReal"(Base := 250.0, Amp := #Amp_TmpC, Lo := #Lo, Hi := #Hi, Seed := #Seed);
	    "ExtDie".TmpAdp002.Act := "FC_NoiseReal"(Base := 249.9, Amp := #Amp_TmpC, Lo := #Lo, Hi := #Hi, Seed := #Seed);
	    "ExtDie".TmpAdp002.Y := "FC_NoiseReal"(Base := 45.0, Amp := #Amp_Y_Pct, Lo := #Lo, Hi := #Hi, Seed := #Seed);

	    // =========================
	    // Zone 1 .. 7 (base dari gambar)
	    // =========================
	    // Zone 1: Set 250.0 / Act 250.1 / Y 55.0
	    "ExtDie".TmpZon001.Set := "FC_NoiseReal"(Base := 250.0, Amp := #Amp_TmpC, Lo := #Lo, Hi := #Hi, Seed := #Seed);
	    "ExtDie".TmpZon001.Act := "FC_NoiseReal"(Base := 250.1, Amp := #Amp_TmpC, Lo := #Lo, Hi := #Hi, Seed := #Seed);
	    "ExtDie".TmpZon001.Y := "FC_NoiseReal"(Base := 55.0, Amp := #Amp_Y_Pct, Lo := #Lo, Hi := #Hi, Seed := #Seed);

	    // Zone 2: Set 250.0 / Act 250.1 / Y 20.0
	    "ExtDie".TmpZon002.Set := "FC_NoiseReal"(Base := 250.0, Amp := #Amp_TmpC, Lo := #Lo, Hi := #Hi, Seed := #Seed);
	    "ExtDie".TmpZon002.Act := "FC_NoiseReal"(Base := 250.1, Amp := #Amp_TmpC, Lo := #Lo, Hi := #Hi, Seed := #Seed);
	    "ExtDie".TmpZon002.Y := "FC_NoiseReal"(Base := 20.0, Amp := #Amp_Y_Pct, Lo := #Lo, Hi := #Hi, Seed := #Seed);

	    // Zone 3: Set 250.0 / Act 250.0 / Y 6.0
	    "ExtDie".TmpZon003.Set := "FC_NoiseReal"(Base := 250.0, Amp := #Amp_TmpC, Lo := #Lo, Hi := #Hi, Seed := #Seed);
	    "ExtDie".TmpZon003.Act := "FC_NoiseReal"(Base := 250.0, Amp := #Amp_TmpC, Lo := #Lo, Hi := #Hi, Seed := #Seed);
	    "ExtDie".TmpZon003.Y := "FC_NoiseReal"(Base := 6.0, Amp := #Amp_Y_Pct, Lo := #Lo, Hi := #Hi, Seed := #Seed);

	    // Zone 4: Set 250.0 / Act 250.0 / Y 0.0
	    "ExtDie".TmpZon004.Set := "FC_NoiseReal"(Base := 250.0, Amp := #Amp_TmpC, Lo := #Lo, Hi := #Hi, Seed := #Seed);
	    "ExtDie".TmpZon004.Act := "FC_NoiseReal"(Base := 250.0, Amp := #Amp_TmpC, Lo := #Lo, Hi := #Hi, Seed := #Seed);
	    "ExtDie".TmpZon004.Y := "FC_NoiseReal"(Base := 0.0, Amp := #Amp_Y_Pct, Lo := #Lo, Hi := #Hi, Seed := #Seed);

	    // Zone 5: Set 250.0 / Act 249.9 / Y 7.0
	    "ExtDie".TmpZon005.Set := "FC_NoiseReal"(Base := 250.0, Amp := #Amp_TmpC, Lo := #Lo, Hi := #Hi, Seed := #Seed);
	    "ExtDie".TmpZon005.Act := "FC_NoiseReal"(Base := 249.9, Amp := #Amp_TmpC, Lo := #Lo, Hi := #Hi, Seed := #Seed);
	    "ExtDie".TmpZon005.Y := "FC_NoiseReal"(Base := 7.0, Amp := #Amp_Y_Pct, Lo := #Lo, Hi := #Hi, Seed := #Seed);

	    // Zone 6: Set 250.0 / Act 250.0 / Y 17.0
	    "ExtDie".TmpZon006.Set := "FC_NoiseReal"(Base := 250.0, Amp := #Amp_TmpC, Lo := #Lo, Hi := #Hi, Seed := #Seed);
	    "ExtDie".TmpZon006.Act := "FC_NoiseReal"(Base := 250.0, Amp := #Amp_TmpC, Lo := #Lo, Hi := #Hi, Seed := #Seed);
	    "ExtDie".TmpZon006.Y := "FC_NoiseReal"(Base := 17.0, Amp := #Amp_Y_Pct, Lo := #Lo, Hi := #Hi, Seed := #Seed);

	    // Zone 7: Set 250.0 / Act 250.1 / Y 57.0
	    "ExtDie".TmpZon007.Set := "FC_NoiseReal"(Base := 250.0, Amp := #Amp_TmpC, Lo := #Lo, Hi := #Hi, Seed := #Seed);
	    "ExtDie".TmpZon007.Act := "FC_NoiseReal"(Base := 250.1, Amp := #Amp_TmpC, Lo := #Lo, Hi := #Hi, Seed := #Seed);
	    "ExtDie".TmpZon007.Y := "FC_NoiseReal"(Base := 57.0, Amp := #Amp_Y_Pct, Lo := #Lo, Hi := #Hi, Seed := #Seed);

END_FUNCTION

FUNCTION "FC_Fluct_DB300_SilDos" : Void
{ S7_Optimized_Access := 'TRUE' }
VERSION : 0.1
// ============================================================
// FLUCTUATION DB300 (SilDos)
// ============================================================
   VAR_INPUT
      Enable : Bool;   // amplitudo fluktuasi per jenis nilai
      Amp_RatioPct : Real;   // Â±0.5 %
      Amp_FdgKgh : Real;   // Â±5.0 kg/h
      Amp_WeiKg : Real;   // Â±1.0 kg
      Amp_LvlKg : Real;   // Â±0.5 kg
      Amp_Y_Pct : Real;   // Â±1.0 %
   END_VAR

   VAR_IN_OUT
      Seed : DInt;
   END_VAR

   VAR_TEMP
      Lo : Real;
      Hi : Real;
   END_VAR


BEGIN
	    IF NOT #Enable THEN
	        RETURN;
	    END_IF;

	    #Lo := -3.4E38;
	    #Hi := 3.4E38;

	    // =========================
	    // Dosing 1
	    // =========================
	    "SilDos".Dos001.RatAct := "FC_NoiseReal"(Base := 0.0, Amp := #Amp_RatioPct, Lo := #Lo, Hi := #Hi, Seed := #Seed);
	    "SilDos".Dos001.FdgAct := "FC_NoiseReal"(Base := 0.0, Amp := #Amp_FdgKgh, Lo := #Lo, Hi := #Hi, Seed := #Seed);
	    "SilDos".Dos001.FdgSet := "FC_NoiseReal"(Base := 0.6, Amp := #Amp_FdgKgh, Lo := #Lo, Hi := #Hi, Seed := #Seed);
	    "SilDos".Dos001.WeiAct := "FC_NoiseReal"(Base := 67.5, Amp := #Amp_WeiKg, Lo := #Lo, Hi := #Hi, Seed := #Seed);

	    // =========================
	    // Dosing 2
	    // =========================
	    "SilDos".Dos002.RatAct := "FC_NoiseReal"(Base := 82.0, Amp := #Amp_RatioPct, Lo := #Lo, Hi := #Hi, Seed := #Seed);
	    "SilDos".Dos002.FdgAct := "FC_NoiseReal"(Base := 982.0, Amp := #Amp_FdgKgh, Lo := #Lo, Hi := #Hi, Seed := #Seed);
	    "SilDos".Dos002.FdgSet := "FC_NoiseReal"(Base := 1013.0, Amp := #Amp_FdgKgh, Lo := #Lo, Hi := #Hi, Seed := #Seed);
	    "SilDos".Dos002.WeiAct := "FC_NoiseReal"(Base := 51.5, Amp := #Amp_WeiKg, Lo := #Lo, Hi := #Hi, Seed := #Seed);

	    // =========================
	    // Dosing 3
	    // =========================
	    "SilDos".Dos003.RatAct := "FC_NoiseReal"(Base := 3.0, Amp := #Amp_RatioPct, Lo := #Lo, Hi := #Hi, Seed := #Seed);
	    "SilDos".Dos003.FdgAct := "FC_NoiseReal"(Base := 35.9, Amp := #Amp_FdgKgh, Lo := #Lo, Hi := #Hi, Seed := #Seed);
	    "SilDos".Dos003.FdgSet := "FC_NoiseReal"(Base := 37.6, Amp := #Amp_FdgKgh, Lo := #Lo, Hi := #Hi, Seed := #Seed);
	    "SilDos".Dos003.WeiAct := "FC_NoiseReal"(Base := 8.7, Amp := #Amp_WeiKg, Lo := #Lo, Hi := #Hi, Seed := #Seed);

	    // =========================
	    // Dosing 4
	    // =========================
	    "SilDos".Dos004.RatAct := "FC_NoiseReal"(Base := 15.0, Amp := #Amp_RatioPct, Lo := #Lo, Hi := #Hi, Seed := #Seed);
	    "SilDos".Dos004.FdgAct := "FC_NoiseReal"(Base := 179.6, Amp := #Amp_FdgKgh, Lo := #Lo, Hi := #Hi, Seed := #Seed);
	    "SilDos".Dos004.FdgSet := "FC_NoiseReal"(Base := 176.1, Amp := #Amp_FdgKgh, Lo := #Lo, Hi := #Hi, Seed := #Seed);
	    "SilDos".Dos004.WeiAct := "FC_NoiseReal"(Base := 20.5, Amp := #Amp_WeiKg, Lo := #Lo, Hi := #Hi, Seed := #Seed);

	    // =========================
	    // Dosing Global
	    // =========================
	    "SilDos".DosGbl.FdgAct := "FC_NoiseReal"(Base := 1227.3, Amp := #Amp_FdgKgh, Lo := #Lo, Hi := #Hi, Seed := #Seed);
	    "SilDos".DosGbl.CmpAct := "FC_NoiseReal"(Base := 96505.7, Amp := (#Amp_WeiKg * 10.0), Lo := #Lo, Hi := #Hi, Seed := #Seed);

	    // =========================
	    // Level Control
	    // =========================
	    "SilDos".LvlCtl.Act := "FC_NoiseReal"(Base := 90.0, Amp := #Amp_LvlKg, Lo := #Lo, Hi := #Hi, Seed := #Seed);
	    "SilDos".LvlCtl.Set := "FC_NoiseReal"(Base := 90.0, Amp := #Amp_LvlKg, Lo := #Lo, Hi := #Hi, Seed := #Seed);
	    "SilDos".LvlCtl.Y := "FC_NoiseReal"(Base := 60.2, Amp := #Amp_Y_Pct, Lo := #Lo, Hi := #Hi, Seed := #Seed);

	    // PmtLvlCtl
	    "SilDos".PmtLvlCtl.Y := "FC_NoiseReal"(Base := 60.2, Amp := #Amp_Y_Pct, Lo := #Lo, Hi := #Hi, Seed := #Seed);
END_FUNCTION

DATA_BLOCK "DB_Sim"
{ S7_Optimized_Access := 'TRUE' }
VERSION : 0.1
NON_RETAIN
// ============================================================
// DB SIM (seed global)
// ============================================================
   VAR
      Seed_All : DInt;
   END_VAR


BEGIN
   Seed_All := 123_456_789;

END_DATA_BLOCK

DATA_BLOCK "FC_Fluct_DB330_Win_DB"
{ S7_Optimized_Access := 'TRUE' }
VERSION : 0.2
NON_RETAIN
"FC_Fluct_DB330_Win"

BEGIN

END_DATA_BLOCK

FUNCTION "FC_Fluct_Master" : Void
{ S7_Optimized_Access := 'TRUE' }
VERSION : 0.3
// ============================================================
// MASTER FC (panggil semua area/DB) - always enable semua DB
// ============================================================
   VAR_INPUT
      Enable : Bool;   // global enable saja
   END_VAR

   VAR_IN_OUT
      Seed : DInt;
   END_VAR


BEGIN
	    IF NOT #Enable THEN
	        RETURN;
	    END_IF;

	    "FC_Fluct_DB300_SilDos"(
	                            Enable := TRUE,
	                            Amp_RatioPct := 0.5,
	                            Amp_FdgKgh := 5.0,
	                            Amp_WeiKg := 1.0,
	                            Amp_LvlKg := 0.5,
	                            Amp_Y_Pct := 1.0,
	                            Seed := #Seed
	    );

	    "FC_Fluct_DB311_ExtMel"(
	                            Enable := TRUE,
	                            Amp_PowKw := 0.2,
	                            Amp_SpdRpm := 1.5,
	                            Amp_TmpC := 0.8,
	                            Amp_PrsBar := 0.3,
	                            Amp_Y_Pct := 1.0,
	                            Seed := #Seed
	    );

	    "FC_Fluct_DB312_ExtMet"(
	                            Enable := TRUE,
	                            Amp_PowKw := 0.2,
	                            Amp_SpdRpm := 1.5,
	                            Amp_TmpC := 0.8,
	                            Amp_Y_Pct := 1.0,
	                            Amp_PrsBar := 0.3,
	                            Seed := #Seed
	    );

	    "FC_Fluct_DB313_ExtFil"(
	                            Enable := TRUE,
	                            Amp_TmpC := 0.8,
	                            Amp_PrsBar := 0.3,
	                            Amp_Y_Pct := 1.0,
	                            Seed := #Seed
	    );

	    "FC_Fluct_DB314_ExtDie"(
	                            Enable := TRUE,
	                            Amp_TmpC := 0.8,
	                            Amp_Y_Pct := 1.0,
	                            Seed := #Seed
	    );

	    "FC_Fluct_DB315_ExtDieBlt"(
	                               Enable := TRUE,
	                               Amp_TmpC := 0.8,
	                               Seed := #Seed
	    );

	    "FC_Fluct_DB316_ExtCox001"(
	                               Enable := TRUE,
	                               Amp_PowKw := 0.2,
	                               Amp_SpdRpm := 1.5,
	                               Amp_LoaPct := 1.0,
	                               Amp_TmpC := 0.8,
	                               Amp_PrsBar := 0.3,
	                               Amp_Y_Pct := 1.0,
	                               Seed := #Seed
	    );

	    "FC_Fluct_DB317_ExtCox002"(
	                               Enable := TRUE,
	                               Amp_PowKw := 0.2,
	                               Amp_SpdRpm := 1.5,
	                               Amp_TmpC := 0.8,
	                               Amp_PrsBar := 0.3,
	                               Amp_Y_Pct := 1.0,
	                               Amp_LoaPct := 1.0,
	                               Seed := #Seed
	    );

	    "FC_Fluct_DB321_StrCas"(
	                            Enable := TRUE,
	                            Amp_SpdPct := 1.0,
	                            Amp_PrsMbar := 5.0,
	                            Amp_TmpC := 0.8,
	                            Amp_Y_Pct := 1.0,
	                            Amp_SpdMpm := 0.3,
	                            Amp_LoaPct := 0.5,
	                            Seed := #Seed
	    );

	    "FC_Fluct_DB322_StrMdo"(
	                            Enable := TRUE,
	                            Amp_TmpC := 0.8,
	                            Amp_Y_Pct := 1.0,
	                            Amp_SpdMpm := 0.5,
	                            Amp_LoaPct := 1.0,
	                            Seed := #Seed
	    );

	    "FC_Fluct_DB323_324_TdoInlMid"(
	                                   Enable := TRUE,
	                                   Amp_TmpC := 0.8,
	                                   Amp_Y_Pct := 1.0,
	                                   Seed := #Seed
	    );

	    "FC_Fluct_DB325_StrTdoOut"(
	                               Enable := TRUE,
	                               Amp_TmpC := 0.8,
	                               Amp_Y_Pct := 1.0,
	                               Amp_SpdMpm := 0.8,
	                               Amp_Loa_Pct := 1.0,
	                               Seed := #Seed
	    );

	    "FC_Fluct_DB326_StrPur"(
	                            Enable := TRUE,
	                            Amp_TmpC := 0.8,
	                            Amp_Y_Pct := 1.0,
	                            Amp_SpdMpm := 0.8,
	                            Amp_LoaPct := 0.5,
	                            Amp_PowKw := 0.2,
	                            Amp_CorSpd := 5,
	                            Seed := #Seed
	    );

	    //"FC_Fluct_DB330_Win"

END_FUNCTION

ORGANIZATION_BLOCK "Cyclic interrupt"
{ S7_Optimized_Access := 'FALSE' }
VERSION : 0.1
   VAR_TEMP
      EV_CLASS : Byte;   // Bits 0-3 = 1:Coming event, Bits 4-7 = 1:Event class 1
      STRT_INF : Byte;   // Start information
      PRIORITY : Byte;   // Priority of OB Execution
      OB_NUMBR : Byte;   // OB number
      RESERVED_1 : Byte;   // Reserved for system
      RESERVED_2 : Byte;   // Reserved for system
      PHS_OFFSET : Int;   // Phase offset
      RESERVED_3 : Int;   // Reserved for system
      EXC_FREQ : Int;   // Frequency of execution
      DATE_TIME : Date_And_Time;   // Date and time OB started
   END_VAR


BEGIN
	"FC_Fluct_Master"(Enable := TRUE,
	                  Seed := "DB_Sim".Seed_All);
	"FC_Fluct_DB330_Win_DB"(
	                        Enable     := TRUE,
	                        Amp_SpdMpm := 0.8,
	                        Amp_LoaPct := 0.5,
	                        Amp_PowKw  := 0.2,
	                        Amp_TmpC   := 0.8,
	                        Amp_TenNm  := 2.0,
	                        Amp_PrsN   := 10.0,
	                        Amp_PosMm  := 0.5,
	                        Seed       := "MD100"
	);

END_ORGANIZATION_BLOCK

